			IF	(((bScrew1Found OR (bScrew1MinFound AND lrPackageThreadTimes = 1)) AND mcScrewer1Stop.Done) OR NOT bRun1 OR mcScrewer1MoveRelative.Done) AND
				(((bScrew2Found OR (bScrew2MinFound AND lrPackageThreadTimes = 1)) AND mcScrewer2Stop.Done) OR NOT bRun2 OR mcScrewer2MoveRelative.Done)
			THEN
				 mcScrewer1MoveRelative.Execute 	:=	FALSE;
				 mcScrewer1Stop.Execute				:=	FALSE;
				 mcScrewer2MoveRelative.Execute 	:=	FALSE;		
				 mcScrewer2Stop.Execute				:=	FALSE;	 
				 iFindingScrewCASE					:=	iFindingScrewCASE	+	10;	
			END_IF
			
		50: 
			IF tonFindingScrewDelay.Q THEN
 				iFindingScrewCASE					:=	iFindingScrewCASE	+	10;						
			END_IF

		60:
			lrStartPosition1						:=	Screwing1AxisRef.NcToPlc.ActPos;
			lrStartPosition2						:=	Screwing2AxisRef.NcToPlc.ActPos;
			iFindingScrewCASE 						:=	0;
			eRunningState							:=	E_GripperScrewer.eScrewing;
			IF bOptionFindScrewInPushingPosition THEN // Opcja - szukanie gwintu w pozycji docisku
				// Przejście do pozycji zakręcania, dlatego że był w pozycji docisku
				eRunningState							:=	E_GripperScrewer.eToScrewingPosition;
			END_IF
		END_CASE
END_IF
END_ACTION

ACTION Running6ScrewingMomentaryMode:
				(********** TRYB MOMENTOWY **********)
					CASE iScrewingCase OF 	
					0:
						(* Wersja 2 - gearowanie Multi Master***************************************************************) 
						IF iTool <> 2 THEN
							bGripper1Actuator						:=	bRun1; // Ponowne załączanie chwytaków, dlatego
							bGripper2Actuator						:=	bRun2; // że jest możliwa duża ilość opcji
						ELSE
							bGripper1Actuator						:=	FALSE; // Ponowne załączanie chwytaków, dlatego
							bGripper2Actuator						:=	FALSE;
						END_IF
						mcHeightGearInMultiMaster.Enable			:=	TRUE;				
						(* Start zakręcania *)
						IF	mcHeightGearInMultiMaster.InGear AND 
							(tonGripper1Delay.Q OR sTool = 'ksztaltowa/do kulek' OR NOT bRun1) AND (tonGripper2Delay.Q OR sTool = 'ksztaltowa/do kulek'  OR NOT bRun2) // ton'y powinny być już wczesniej załączone jeżeli były chwytaki	
						THEN

							mcScrewer1TorqueControl.Execute					:=	bRun1;
							mcScrewer1TorqueControl.Torque					:=	5000;//(INT_TO_UINT(iScrewer1SetTorque+3)*10)+iScrewer1AddTorque;	
							mcScrewer1TorqueControl.TorqueRamp				:=	4000;
							mcScrewer1TorqueControl.VelocityLimitHigh		:=	10;							
							mcScrewer1TorqueControl.VelocityLimitLow		:=	-5000;//(lrScrewerSpeed);
												
							mcScrewer2TorqueControl.Execute					:=	bRun2;
							mcScrewer2TorqueControl.Torque					:=	5000;//(INT_TO_UINT(iScrewer2SetTorque+3)*10)+iScrewer2AddTorque;	
							mcScrewer2TorqueControl.TorqueRamp				:=	4000;
							mcScrewer2TorqueControl.VelocityLimitHigh		:=	10;							
							mcScrewer2TorqueControl.VelocityLimitLow		:=	-5000;//(lrScrewerSpeed);
	
							iScrewingCase									:=	iScrewingCase + 10;			
						END_IF
						
					10:	
					
						IF ABS(ABS(lrStartPosition1)-ABS(Screwing1AxisRef.NcToPlc.ActPos))>(lrPackageTurnoversToFullScrewed*360.0/7)  THEN 
							mcScrewer1TorqueControl.Torque					:=	-9;		
							mcScrewer1TorqueControl.TorqueRamp				:=	1500;					
							mcScrewer1TorqueControl.VelocityLimitLow		:=	-4000;
						END_IF	
							
						IF ABS(ABS(lrStartPosition2)-ABS(Screwing2AxisRef.NcToPlc.ActPos))>(lrPackageTurnoversToFullScrewed*360.0/7)  THEN 
							mcScrewer2TorqueControl.Torque					:=	-9;		
							mcScrewer2TorqueControl.TorqueRamp				:=	1500;					
							mcScrewer2TorqueControl.VelocityLimitLow		:=	-4000;
						END_IF	
						
						IF ABS(ABS(lrStartPosition1)-ABS(Screwing1AxisRef.NcToPlc.ActPos))>(lrPackageTurnoversToFullScrewed*360.0/6)  THEN 
							mcScrewer1TorqueControl.Torque					:=	(INT_TO_UINT(iScrewer1SetTorque)+iScrewer1AddTorque);		
							mcScrewer1TorqueControl.TorqueRamp				:=	4000;					
							mcScrewer1TorqueControl.VelocityLimitLow		:=	-(lrScrewerSpeed);
						END_IF	
							
						IF ABS(ABS(lrStartPosition2)-ABS(Screwing2AxisRef.NcToPlc.ActPos))>(lrPackageTurnoversToFullScrewed*360.0/6)  THEN 
							mcScrewer2TorqueControl.Torque					:=	(INT_TO_UINT(iScrewer2SetTorque)+iScrewer2AddTorque);		
							mcScrewer2TorqueControl.TorqueRamp				:=	4000;					
							mcScrewer2TorqueControl.VelocityLimitLow		:=	-(lrScrewerSpeed);
						END_IF						
						(*IF tonMomentaryScrewing1Timer.Q OR bWarning1 THEN
							mcScrewer1Stop.Execute				:=	TRUE;
							bGripper1Actuator					:=	FALSE;
							mcScrewer1TorqueControl.Execute		:=	FALSE;
							uiScrewing1TorqueControl			:=	0;
							bScrewed1							:=	TRUE;	
						END_IF
						IF tonMomentaryScrewing2Timer.Q OR bWarning2 THEN
							mcScrewer2Stop.Execute				:=	TRUE;
							bGripper2Actuator					:=	FALSE;
							mcScrewer2TorqueControl.Execute		:=	FALSE;
							uiScrewing2TorqueControl			:=	0;
							bScrewed2							:=	TRUE;		
						END_IF*)
								
						IF tonMomentaryScrewing1Timer.Q OR bWarning1 THEN
							bGripper1Actuator					:=	FALSE;
							bScrewed1							:=	TRUE;	
						END_IF
						IF tonMomentaryScrewing2Timer.Q OR bWarning2 THEN
							bGripper2Actuator					:=	FALSE;
							bScrewed2							:=	TRUE;		
						END_IF
				
						IF tonTightScrewing1TimerAndOpenedGripper.Q OR bWarning1 THEN
							mcScrewer1Stop.Execute				:=	TRUE;
							mcScrewer1TorqueControl.Execute		:=	FALSE;
						END_IF
						IF tonTightScrewing2TimerAndOpenedGripper.Q OR bWarning2 THEN
							mcScrewer2Stop.Execute				:=	TRUE;
							mcScrewer2TorqueControl.Execute		:=	FALSE;
						END_IF											
				
						// Warunki zakręcenia zaleznie od uruchomionej zakręcarki
//						IF (bScrewed1 OR NOT bRun1) AND (bScrewed2 OR NOT bRun2) AND
//							(mcScrewer1Stop.Done OR NOT mcScrewer1Stop.Execute) AND 
//							(mcScrewer2Stop.Done OR NOT mcScrewer2Stop.Execute) THEN
						IF (tonTightScrewing1TimerAndOpenedGripper.Q OR NOT bRun1) AND (tonTightScrewing2TimerAndOpenedGripper.Q OR NOT bRun2) AND
							(mcScrewer1Stop.Done OR NOT mcScrewer1Stop.Execute) AND 
							(mcScrewer2Stop.Done OR NOT mcScrewer2Stop.Execute) THEN
								mcScrewer1Stop.Execute			:= FALSE;
								mcScrewer2Stop.Execute			:= FALSE;
								iScrewingCase					:= iScrewingCase + 10;		
						END_IF
					20:
						(* Rozgearowanie osi *)
						mcHeightGearOut.Execute				:=	TRUE;
						mcHeightGearInMultiMaster.Enable	:=	FALSE;
	
						IF  mcHeightGearOut.Done THEN
							mcHeightGearOut.Execute					:= FALSE;
							eRunningState							:= E_GripperScrewer.eHolding;	
							iScrewingCase							:= 0;	
						END_IF			
					END_CASE
END_ACTION

ACTION Running6ScrewingPositionTorqueMode:
				(********* TRYB POZYCYJNY  *********)
				
				lrPackageThreadPitch;	
				(*Wymuszanie zwiększonego momentu przez 1/4 całego zakręcania*)
				IF ABS(ABS(lrStartPosition1)-ABS(Screwing1AxisRef.NcToPlc.ActPos))>(lrPackageTurnoversToFullScrewed*360.0/7)  THEN 
							uiScrewing1TorqueControl			:=	(INT_TO_UINT(iScrewer1SetTorque+3)*10)+(iScrewer1AddTorque*10);	
				ELSE		uiScrewing1TorqueControl			:=	6000;
				END_IF
				//uiScrewing1TorqueControl			:=	(INT_TO_UINT(iScrewerSetTorque+3)*10)+iScrewer1AddTorque;	
				(*Wymuszanie zwiększonego momentu przez 1/4 całego zakręcania*)
				IF ABS(ABS(lrStartPosition2)-ABS(Screwing2AxisRef.NcToPlc.ActPos))>(lrPackageTurnoversToFullScrewed*360.0/7)  THEN 
							uiScrewing2TorqueControl			:=	(INT_TO_UINT(iScrewer2SetTorque+3)*10)+(iScrewer2AddTorque*10);		
				ELSE		uiScrewing2TorqueControl			:=	6000;
				END_IF	

					CASE iScrewingCase OF 	
					0:
						(* Wersja 2 - gearowanie Multi Master***************************************************************) 
						IF iTool <> 2 THEN
							bGripper1Actuator						:=	bRun1; // Ponowne załączanie chwytaków, dlatego
							bGripper2Actuator						:=	bRun2; // że jest możliwa duża ilość opcji
						ELSE
							bGripper1Actuator						:=	FALSE; // Ponowne załączanie chwytaków, dlatego
							bGripper2Actuator						:=	FALSE; // że jest możliwa duża ilość opcji
						END_IF
						mcHeightGearInMultiMaster.Enable			:=	TRUE;				
						(* Start zakręcania *)
						IF	mcHeightGearInMultiMaster.InGear AND 
							(tonGripper1Delay.Q OR sTool = 'ksztaltowa/do kulek' OR NOT bRun1) AND (tonGripper2Delay.Q OR sTool = 'ksztaltowa/do kulek' OR NOT bRun2) // ton'y powinny być już wczesniej załączone jeżeli były chwytaki	
						THEN

							CASE iScrewing2Case OF 	
								
							0:
							
								mcScrewer1MoveVelocity2.Velocity		:=	5000;
								mcScrewer1MoveVelocity2.Execute		:=	bRun1;
								mcScrewer1MoveVelocity2.Direction	:=	MC_Positive_Direction;
																				
								mcScrewer2MoveVelocity2.Velocity		:=	5000;
								mcScrewer2MoveVelocity2.Execute		:=	bRun2;
								mcScrewer2MoveVelocity2.Direction	:=	MC_Positive_Direction;	
	
								iScrewing2Case						:=	iScrewing2Case + 10;										
							
							10:
								mcScrewer1MoveVelocity2.Execute		:=	FALSE;
								mcScrewer2MoveVelocity2.Execute		:=	FALSE;
							
								iScrewing2Case						:=	iScrewing2Case + 10;
	
							20:
							
								mcScrewer1MoveVelocity.Velocity		:=	lrScrewerSpeed;		
								mcScrewer1MoveVelocity.Direction	:=	MC_Positive_Direction;	
								IF ABS(ABS(lrStartPosition1)-ABS(Screwing1AxisRef.NcToPlc.ActPos))>(lrPackageTurnoversToFullScrewed*360.0/7)  THEN 									
									mcScrewer1MoveVelocity.Execute		:=	bRun1;									
								END_IF
								mcScrewer2MoveVelocity.Velocity		:=	lrScrewerSpeed;	
								mcScrewer1MoveVelocity.Direction		:=	MC_Positive_Direction;	
								IF ABS(ABS(lrStartPosition2)-ABS(Screwing2AxisRef.NcToPlc.ActPos))>(lrPackageTurnoversToFullScrewed*360.0/7)  THEN 
	
									mcScrewer2MoveVelocity.Execute		:=	bRun2;
								END_IF			

								IF (mcScrewer1MoveVelocity.Execute OR NOT bRun1) AND (mcScrewer2MoveVelocity.Execute OR NOT bRun2) THEN
									iScrewing2Case					:= 0	;
									iScrewingCase					:= iScrewingCase + 10;		
								END_IF
								
							END_CASE
							
						END_IF
						
					10:	
					
						(*Zmniejszanie prędkości jeżeli jest już przytrzymanie*)
						IF tonTightScrewing1Timer.ET > T#0S AND Screwing1AxisRef.NcToPlc.ActVelo < 10 THEN
							//mcScrewer1MoveVelocity.Execute		:= FALSE;
							//mcScrewer1MoveVelocity2.Execute		:= FALSE;
							
							//mcScrewer1MoveVelocity3.Velocity	:=	10;
							//mcScrewer1MoveVelocity3.Execute		:=	bRun1;
							//mcScrewer1MoveVelocity3.Direction	:=	MC_Positive_Direction;		

							rScrewing1ProportionalGain	:= 0;
							//rScrewing2ProportionalGain	:= 0;												
						END_IF
						
						IF tonTightScrewing2Timer.ET > T#0S AND Screwing2AxisRef.NcToPlc.ActVelo < 10 THEN
							//mcScrewer2MoveVelocity.Execute		:= FALSE;
							//mcScrewer2MoveVelocity2.Execute		:= FALSE;
							
							//mcScrewer2MoveVelocity3.Velocity	:=	10;
							//mcScrewer2MoveVelocity3.Execute		:=	bRun1;
							//mcScrewer2MoveVelocity3.Direction	:=	MC_Positive_Direction;		

							//rScrewing1ProportionalGain	:= 0;
							rScrewing2ProportionalGain	:= 0;												
						END_IF					
					
						(* Sprawdzanie czy osiągnięto moment lub zbyt długie zakracanie*)				
						IF tonTightScrewing1Timer.Q OR bWarning1 THEN
							bGripper1Actuator					:=	FALSE;
							bScrewed1							:=	TRUE;	
						END_IF
						IF tonTightScrewing2Timer.Q OR bWarning2 THEN
							bGripper2Actuator					:=	FALSE;
							bScrewed2							:=	TRUE;		
						END_IF
	
						IF tonTightScrewing1TimerAndOpenedGripper.Q THEN
							mcScrewer1Stop.Execute				:=	TRUE;
							mcScrewer1MoveVelocity.Execute		:=	FALSE;
							mcScrewer1MoveVelocity2.Execute		:=	FALSE;
							mcScrewer1MoveVelocity3.Execute		:=	FALSE;							
							uiScrewing1TorqueControl			:=	0;
						END_IF
						IF tonTightScrewing2TimerAndOpenedGripper.Q THEN
							mcScrewer2Stop.Execute				:=	TRUE;
							mcScrewer2MoveVelocity.Execute		:=	FALSE;
							mcScrewer2MoveVelocity2.Execute		:=	FALSE;	
							mcScrewer2MoveVelocity3.Execute		:=	FALSE;							
							uiScrewing2TorqueControl			:=	0;
						END_IF
					
						// Warunki zakręcenia zaleznie od uruchomionej zakręcarki
						IF (tonTightScrewing1TimerAndOpenedGripper.Q OR NOT bRun1) AND (tonTightScrewing2TimerAndOpenedGripper.Q OR NOT bRun2) AND
							(mcScrewer1Stop.Done OR NOT mcScrewer1Stop.Execute) AND 
							(mcScrewer2Stop.Done OR NOT mcScrewer2Stop.Execute) THEN
								mcScrewer1Stop.Execute			:= FALSE;
								mcScrewer2Stop.Execute			:= FALSE;
								iScrewingCase					:= iScrewingCase + 10;		
						END_IF
						
					20:
						(* Rozgearowanie osi *)
						mcHeightGearOut.Execute				:=	TRUE;
						mcHeightGearInMultiMaster.Enable	:=	FALSE;
	
						IF  mcHeightGearOut.Done THEN
							mcHeightGearOut.Execute					:= FALSE;
							eRunningState							:= E_GripperScrewer.eHolding;	
							iScrewingCase							:= 0;	
						END_IF			
					END_CASE
END_ACTION

ACTION Screwer1ControlBlocks:
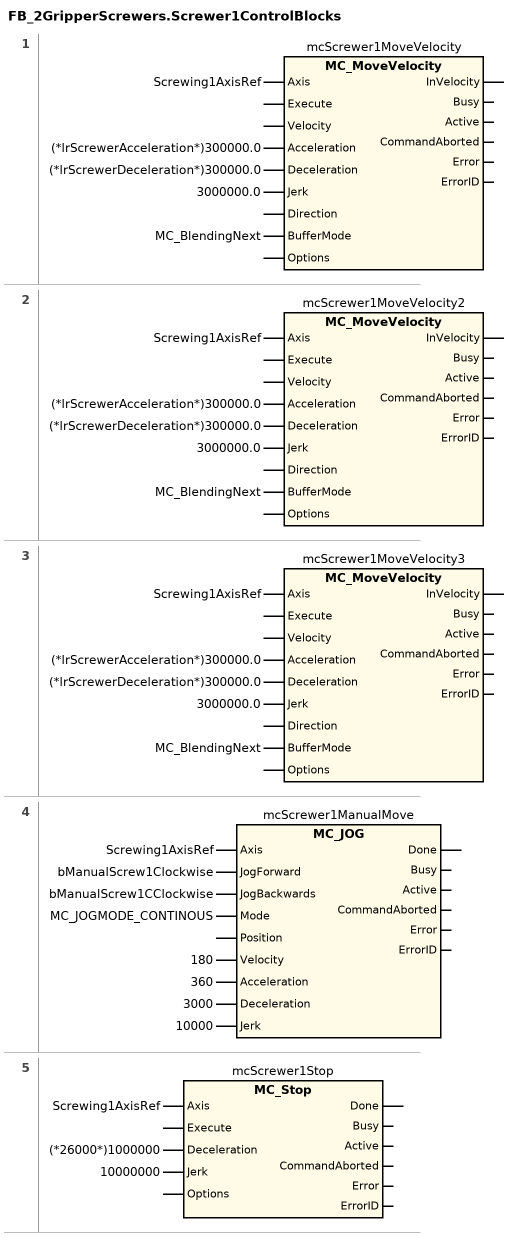
// NETWORK 1
mcScrewer1MoveVelocity(
    Axis := Screwing1AxisRef,
    Acceleration := (*lrScrewerAcceleration*)300000.0,
    Deceleration := (*lrScrewerDeceleration*)300000.0,
    Jerk := 3000000.0,
    BufferMode := MC_BlendingNext); // MC_MoveVelocity

// NETWORK 2
mcScrewer1MoveVelocity2(
    Axis := Screwing1AxisRef,
    Acceleration := (*lrScrewerAcceleration*)300000.0,
    Deceleration := (*lrScrewerDeceleration*)300000.0,
    Jerk := 3000000.0,
    BufferMode := MC_BlendingNext); // MC_MoveVelocity

// NETWORK 3
mcScrewer1MoveVelocity3(
    Axis := Screwing1AxisRef,
    Acceleration := (*lrScrewerAcceleration*)300000.0,
    Deceleration := (*lrScrewerDeceleration*)300000.0,
    Jerk := 3000000.0,
    BufferMode := MC_BlendingNext); // MC_MoveVelocity

// NETWORK 4
mcScrewer1ManualMove(
    Axis := Screwing1AxisRef,
    JogForward := bManualScrew1Clockwise,
    JogBackwards := bManualScrew1CClockwise,
    Mode := MC_JOGMODE_CONTINOUS,
    Velocity := 180,
    Acceleration := 360,
    Deceleration := 3000,
    Jerk := 10000); // MC_JOG

// NETWORK 5
mcScrewer1Stop(Axis := Screwing1AxisRef, Deceleration := (*26000*)1000000, Jerk := 10000000); // MC_Stop

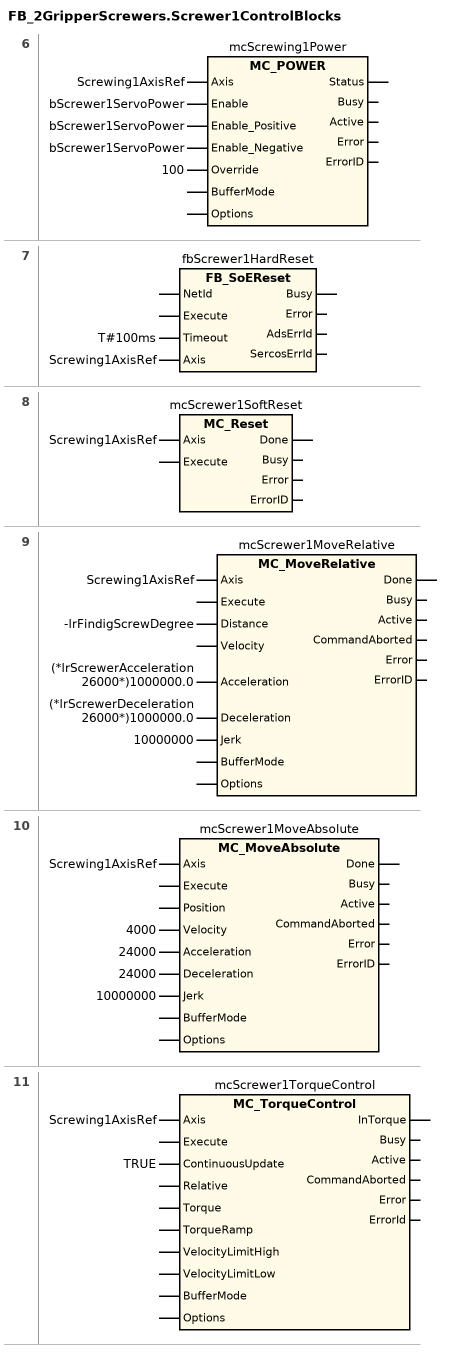
// NETWORK 6
mcScrewing1Power(
    Axis := Screwing1AxisRef,
    Enable := bScrewer1ServoPower,
    Enable_Positive := bScrewer1ServoPower,
    Enable_Negative := bScrewer1ServoPower,
    Override := 100); // MC_POWER

// NETWORK 7
fbScrewer1HardReset(Timeout := T#100ms, Axis := Screwing1AxisRef); // FB_SoEReset

// NETWORK 8
mcScrewer1SoftReset(Axis := Screwing1AxisRef); // MC_Reset

// NETWORK 9
mcScrewer1MoveRelative(
    Axis := Screwing1AxisRef,
    Distance := -lrFindigScrewDegree,
    Acceleration := (*lrScrewerAcceleration 26000*)1000000.0,
    Deceleration := (*lrScrewerDeceleration 26000*)1000000.0,
    Jerk := 10000000); // MC_MoveRelative

// NETWORK 10
mcScrewer1MoveAbsolute(
    Axis := Screwing1AxisRef,
    Velocity := 4000,
    Acceleration := 24000,
    Deceleration := 24000,
    Jerk := 10000000); // MC_MoveAbsolute

// NETWORK 11
mcScrewer1TorqueControl(Axis := Screwing1AxisRef, ContinuousUpdate := TRUE); // MC_TorqueControl

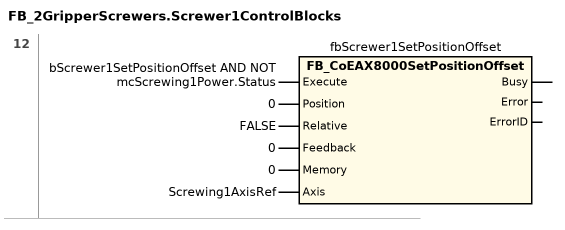
// NETWORK 12
fbScrewer1SetPositionOffset(
    Execute := bScrewer1SetPositionOffset AND NOT mcScrewing1Power.Status,
    Position := 0,
    Relative := FALSE,
    Feedback := 0,
    Memory := 0,
    Axis := Screwing1AxisRef); // FB_CoEAX8000SetPositionOffset
END_ACTION

ACTION Screwer2ControlBlocks:
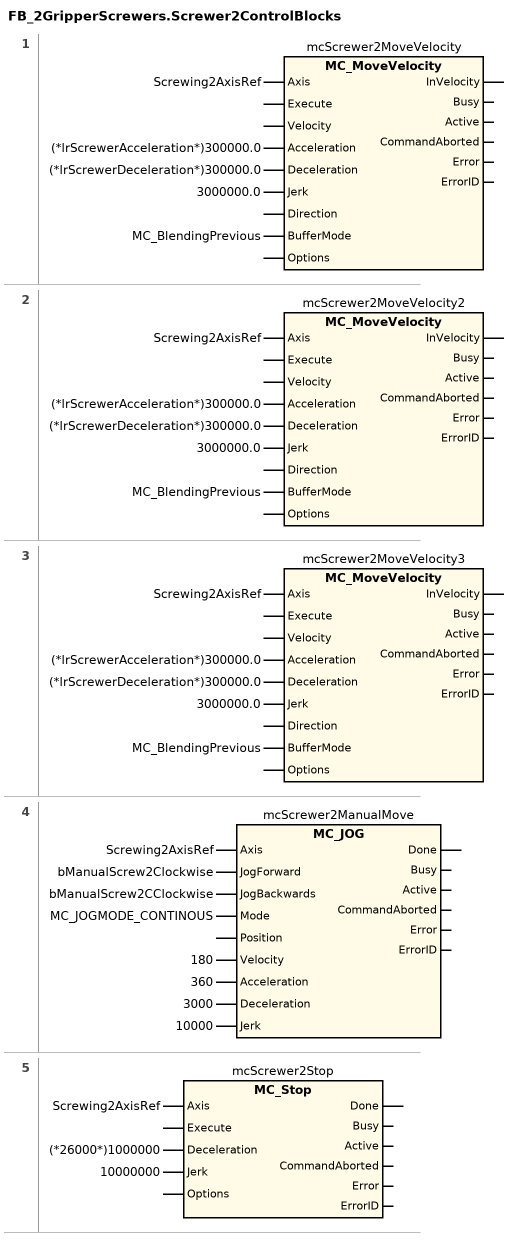
// NETWORK 1
mcScrewer2MoveVelocity(
    Axis := Screwing2AxisRef,
    Acceleration := (*lrScrewerAcceleration*)300000.0,
    Deceleration := (*lrScrewerDeceleration*)300000.0,
    Jerk := 3000000.0,
    BufferMode := MC_BlendingPrevious); // MC_MoveVelocity

// NETWORK 2
mcScrewer2MoveVelocity2(
    Axis := Screwing2AxisRef,
    Acceleration := (*lrScrewerAcceleration*)300000.0,
    Deceleration := (*lrScrewerDeceleration*)300000.0,
    Jerk := 3000000.0,
    BufferMode := MC_BlendingPrevious); // MC_MoveVelocity

// NETWORK 3
mcScrewer2MoveVelocity3(
    Axis := Screwing2AxisRef,
    Acceleration := (*lrScrewerAcceleration*)300000.0,
    Deceleration := (*lrScrewerDeceleration*)300000.0,
    Jerk := 3000000.0,
    BufferMode := MC_BlendingPrevious); // MC_MoveVelocity

// NETWORK 4
mcScrewer2ManualMove(
    Axis := Screwing2AxisRef,
    JogForward := bManualScrew2Clockwise,
    JogBackwards := bManualScrew2CClockwise,
    Mode := MC_JOGMODE_CONTINOUS,
    Velocity := 180,
    Acceleration := 360,
    Deceleration := 3000,
    Jerk := 10000); // MC_JOG

// NETWORK 5
mcScrewer2Stop(Axis := Screwing2AxisRef, Deceleration := (*26000*)1000000, Jerk := 10000000); // MC_Stop

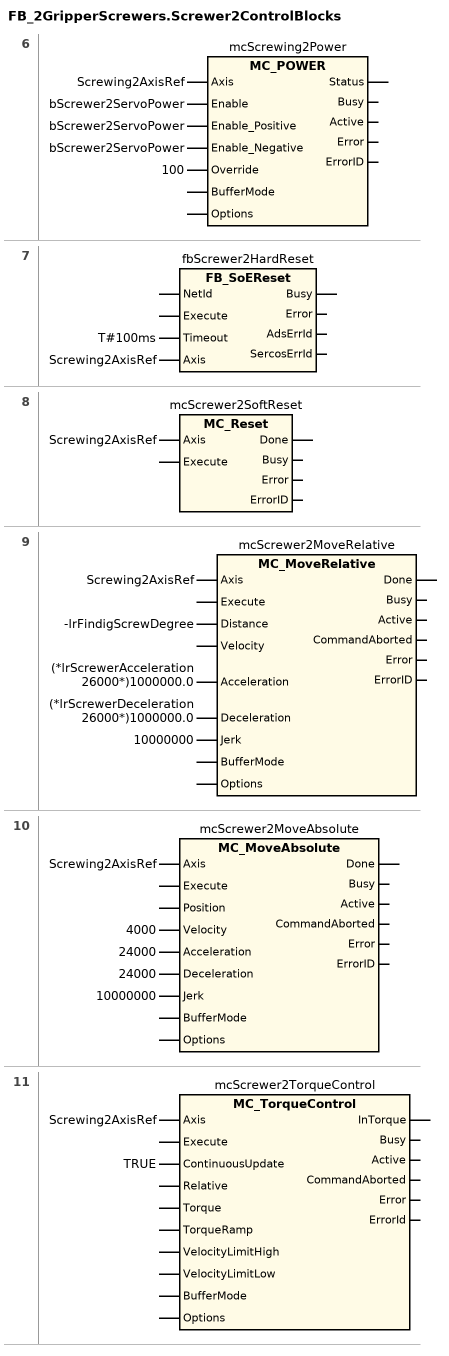
// NETWORK 6
mcScrewing2Power(
    Axis := Screwing2AxisRef,
    Enable := bScrewer2ServoPower,
    Enable_Positive := bScrewer2ServoPower,
    Enable_Negative := bScrewer2ServoPower,
    Override := 100); // MC_POWER

// NETWORK 7
fbScrewer2HardReset(Timeout := T#100ms, Axis := Screwing2AxisRef); // FB_SoEReset

// NETWORK 8
mcScrewer2SoftReset(Axis := Screwing2AxisRef); // MC_Reset

// NETWORK 9
mcScrewer2MoveRelative(
    Axis := Screwing2AxisRef,
    Distance := -lrFindigScrewDegree,
    Acceleration := (*lrScrewerAcceleration 26000*)1000000.0,
    Deceleration := (*lrScrewerDeceleration 26000*)1000000.0,
    Jerk := 10000000); // MC_MoveRelative

// NETWORK 10
mcScrewer2MoveAbsolute(
    Axis := Screwing2AxisRef,
    Velocity := 4000,
    Acceleration := 24000,
    Deceleration := 24000,
    Jerk := 10000000); // MC_MoveAbsolute

// NETWORK 11
mcScrewer2TorqueControl(Axis := Screwing2AxisRef, ContinuousUpdate := TRUE); // MC_TorqueControl

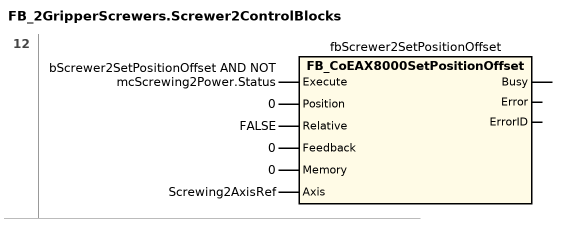
// NETWORK 12
fbScrewer2SetPositionOffset(
    Execute := bScrewer2SetPositionOffset AND NOT mcScrewing2Power.Status,
    Position := 0,
    Relative := FALSE,
    Feedback := 0,
    Memory := 0,
    Axis := Screwing2AxisRef); // FB_CoEAX8000SetPositionOffset
END_ACTION

ACTION Simulation:
(* Przyśpieszanie bloku gdy jest włączona symulacja*)

//tonSimulationScrewing1			(IN:=eRunningState=E_GripperScrewer.eScrewing 	AND bRun1 AND NOT bScrewed1 AND bSimulation,	PT:=T#0MS);
//tonSimulationScrewing2			(IN:=eRunningState=E_GripperScrewer.eScrewing 	AND bRun1 AND NOT bScrewed2 AND bSimulation,	PT:=T#0MS);

IF bSimulation THEN 			// Włączona symulacja
	tTooLongScrewing1 := T#250MS;
	tTooLongScrewing2 := T#250MS;	
ELSE							// Normalna praca
	tTooLongScrewing1 := T#3S; 	//Zmienić na 2
	tTooLongScrewing2 := T#3S;	//Zmienić na 2
END_IF
END_ACTION

ACTION Statistics:

IF LREAL_TO_INT(lrHeightEndScrewingPosition)<> LREAL_TO_INT(lrHeightReadyPosition) THEN
	rtrigCycleTimerRead(CLK:=LREAL_TO_INT(lrHeightActualPosition) = LREAL_TO_INT(lrHeightReadyPosition));
	IF rtrigCycleTimerRead.Q THEN
			tCycleTime:=tonCycleTimer.ET;
	END_IF
	tonCycleTimer(IN:=LREAL_TO_INT(lrHeightActualPosition) <> LREAL_TO_INT(lrHeightReadyPosition),PT:=T#1D);	
ELSE
	rtrigCycleTimerRead(CLK:=(eRunningState=E_GripperScrewer.eDone) OR (eRunningState=E_GripperScrewer.eNotDone));
	IF rtrigCycleTimerRead.Q THEN
		tCycleTime:=tonCycleTimer.ET;
	END_IF
	tonCycleTimer(IN:=eRunningState>E_GripperScrewer.eReady,PT:=T#1D);
END_IF
END_ACTION

ACTION Tools:
(*Narzędzia*)
AsToolDescription[0] := 'Głowica dwuszczękowa';
AsToolDescription[1] := 'Głowica trójszczękowa'; 
AsToolDescription[2] := 'Głowica kształtowa/do kulek';
AsToolDescription[3] := 'Głowica wbijająca'; 
AsToolDescription[4] := 'Głowica zasysająca';


(*Głowica wbijająca*)
IF iTool = 3 THEN
	bOptionCapPushingWithoutScrewing := TRUE;
ELSE
	bOptionCapPushingWithoutScrewing := FALSE;
END_IF

(*Przepisanie wybranego narzędzia do zmiennej typu string*)
(*!!!!! NIE ZMIENIAĆ OPISÓW, POWIĄZANE W PROGRAMIE !!!!!!*)
(* Wysokość narzędzia od pkt. bazowania

		Glowica dwuszczekowa
           |	|
		   |	|
	|------|    |-----|
	|	 _______	  |
	|	|		  |   |
   ||	||		  |   |
   ||	||		  |	  |
   |---- |		  -----	<-pkt. bazowania 	<-|
   |	 |	                                  |
   |	 ---|	  							iToolHeight (mm)
   |druk	|                                 |
   ---------|	  							<-|

*)


IF iTool = 0 THEN sTool := 'dwuszczekowa';			iToolHeight	:=	23;		END_IF 
IF iTool = 1 THEN sTool := 'trojszczekowa';			iToolHeight	:=	-5;	END_IF 
IF iTool = 2 THEN sTool := 'ksztaltowa/do kulek';	iToolHeight	:=	-5;		END_IF 
IF iTool = 3 THEN sTool := 'wbijajaca';				iToolHeight	:=	23;		END_IF 
IF iTool = 4 THEN sTool := 'zasysajaca';			iToolHeight	:=	-4;		END_IF
END_ACTION

ACTION TorqueControl:

(*Konfiguracja MC_TorqueControl*)
//T_TorqueControlOptions;
mcScrewer1TorqueControl.Options.EnableManualTorqueStartValue := TRUE;
mcScrewer1TorqueControl.Options.ManualTorqueStartValue       := Screwing1AxisRef.NcToPlc.ActTorque;

mcScrewer2TorqueControl.Options.EnableManualTorqueStartValue := TRUE;
mcScrewer2TorqueControl.Options.ManualTorqueStartValue       :=  Screwing2AxisRef.NcToPlc.ActTorque;
END_ACTION

ACTION Warnings:
//Resetowanie warningów przy nastepnym cyklu

IF rtRun1.Q  OR rtRun2.Q THEN
	
	bWarning1			:=	FALSE;
	bWarning1A			:=	FALSE;
	bWarning1B			:=	FALSE;
	bWarning1C			:=	FALSE;
	bWarning1D			:=	FALSE;
	bWarning1E			:=	FALSE;	
	bWarning2			:=	FALSE;
	bWarning2A			:=	FALSE;
	bWarning2B			:=	FALSE;
	bWarning2C			:=	FALSE;
	bWarning2D			:=	FALSE;
	bWarning2E			:=	FALSE;
END_IF
END_ACTION

END_FUNCTION_BLOCK

// ---- POUs/FB/POUsAxisOnline/AX8000/FB_McAxisOnlineAX8000.TcPOU
//==================================================================================================
//							Beckhoff Automation Poland
//									7.12.2018
//	Wszystkomajacy blok funkcyjny do sterowania osia, 
//	wymagane biblioteki: Tc2_EtherCAT, Tc2_MC2_Drive, Tc2_MC2
//  v1.5	|| TC v 3.1.4022.27		|| - dodane opisy bledow w formie zmiennych typu string
// 	v1.4 	|| TC v 3.1.4022.20	 	|| - ACT_MotorMonitoring - only for real axis
// 	v1.3 	|| TC v 3.1.4022.16	 	|| - spojne z AX5000
// 	v1.2 	|| TC v 3.1.4022.16	 	|| - Added ACT_SetPositionIO, migration part of logic from ACT_SetPosition to ACT_SetPositionIO
// 	v1.1 	|| TC v 3.1.4022.16	 	|| - ACT_MotorMonitoring - is executing always, ACT_Initialization - optimalization
// 	v1.0 	|| TC v 3.1.4022.16	 	|| - first edition
//==================================================================================================
{attribute 'reflection'}
FUNCTION_BLOCK FB_McAxisOnlineAX8000
VAR_IN_OUT
	stMcAxisOnline						: ST_McAxisOnline;
	Axis								: AXIS_REF;
END_VAR
VAR
	mcPower								: MC_Power;
	mcStop								: MC_Stop;
	mcHalt								: MC_Halt;
	mcStopSS1							: MC_Stop;
	mcStopSS2							: MC_Stop;
	mcReset								: MC_Reset;
	mcHome								: MC_Home;
	mcSetPosition						: MC_SetPosition;
	fbSetPositionOffset					: FB_CoEAX8000SetPositionOffset;
	mcJog								: MC_Jog;

	mcMoveAbsolute						: MC_MoveAbsolute;
	mcMoveRelative						: MC_MoveRelative;
	mcMoveVelocity						: MC_MoveVelocity;
	mcMoveModulo						: MC_MoveModulo;
	mcMoveAbsolute2						: MC_MoveAbsolute;
	mcMoveRelative2						: MC_MoveRelative;
	mcMoveVelocity2						: MC_MoveVelocity;
	mcMoveModulo2						: MC_MoveModulo;

	fbMotorMonitoring					: FB_MotorMonitoringAX8000;
	fbHoldingBrakeCtrl					: FB_HoldingBrakeCtrlAX8000;
	fbNcLimitSwitch						: FB_NcSWLimitSwitchCtrl;
	tonGetDriveDiag						: TON;
	fbReadChannelErrorCode				: FB_ReadChannelErrorCodeAX8000;
	
	mcReadDriveAddress					: MC_ReadDriveAddress;
	mcReadParameterSet					: MC_ReadParameterSet;
	fbGetDriveRef						: FB_GetDriveRef;

	// Internal
	bInitialized						: BOOL;
	bCommError							: BOOL;
	bReadParameterError					: BOOL;
	bInitError							: BOOL;
	bDriveError							: BOOL;
	bFBError							: BOOL;
	
// Initialization
	iInitStep							: INT;
	bInitializationError				: BOOL;
	wInitializationErrorCounter			: WORD;
	bDriveAddressReady					: BOOL;
	bDriveRefReady						: BOOL;
	bReadParameterSetReady				: BOOL;
	tonDelay							: TON;
// Re init
	udiOnlineChangeCntOld				: UDINT;
	bOnlineChangeDetected				: BOOL;
	bReInit								: BOOL;
	bReInitialized						: BOOL;
	bReInitializationError				: BOOL;
	{attribute 'instance-path'}
	{attribute 'noinit'}
	sInstancePath						: STRING;
END_VAR

// Device dependent initialization 
ACT_Initialization();
// Device independent commands, mostly NC 
ACT_States();
ACT_SWLimitSwitch();
ACT_Stop();
ACT_Power();
ACT_Homing();
ACT_Jog();
ACT_Move();
ACT_Reset();
ACT_SetPosition();
// Device dependent commands
// Motor monitoring possible only with real axis
IF NOT Axis.Status.OpMode.SimulationAxis THEN
	ACT_MotorMonitoring();
END_IF
// Device dependent commands, possible only on real axis after complete initialization
IF bInitialized AND NOT Axis.Status.OpMode.SimulationAxis THEN
	ACT_SetPositionIO();
	ACT_DriveDiag();
	ACT_HoldingBrakeCtrl();
END_IF

// Device independent error collection
ACT_ErrorCollection();

ACTION ACT_DriveDiag:
// Auto update when drive error
tonGetDriveDiag(IN:= stMcAxisOnline.stError.bDriveError AND NOT tonGetDriveDiag.Q, PT:= T#5S, Q=> , ET=> );

fbReadChannelErrorCode(	bExecute				:= stMcAxisOnline.stChannelErrorCode.bExecute OR tonGetDriveDiag.Q,
						stDriveRef				:= stMcAxisOnline.stDriveRef,
						bBusy					=> stMcAxisOnline.stChannelErrorCode.bBusy,
						bError					=> stMcAxisOnline.stChannelErrorCode.bError,
						iAdsErrId				=> stMcAxisOnline.stChannelErrorCode.uiAdsErrId,
						iCANopenErrId			=> stMcAxisOnline.stChannelErrorCode.uiSecErrId,
						uiChannelErrorCode		=> stMcAxisOnline.stChannelErrorCode.uiChannelErrorCode,
						uiChannelErrorCodeHex	=> stMcAxisOnline.stChannelErrorCode.uiChannelErrorCodeHex);
END_ACTION

ACTION ACT_ErrorCollection:
// Error flags
stMcAxisOnline.stError.bDriveError					:= Axis.Status.DriveDeviceError;

stMcAxisOnline.stError.bNcError						:= Axis.Status.Error;

stMcAxisOnline.stError.bFBError						:= stMcAxisOnline.mcPower.bError OR stMcAxisOnline.mcReset.bError OR stMcAxisOnline.mcHome.bError OR stMcAxisOnline.mcJog.bError
													OR stMcAxisOnline.mcHalt.bError OR stMcAxisOnline.mcStop.bError OR stMcAxisOnline.mcSS1.bError OR stMcAxisOnline.mcSS2.bError
													OR stMcAxisOnline.mcMoveAbsolute.bError OR stMcAxisOnline.mcMoveRelative.bError OR stMcAxisOnline.mcMoveVelocity.bError OR stMcAxisOnline.mcMoveModulo.bError
													OR stMcAxisOnline.mcMoveAbsolute2.bError OR stMcAxisOnline.mcMoveRelative2.bError OR stMcAxisOnline.mcMoveVelocity2.bError OR stMcAxisOnline.mcMoveModulo2.bError
													OR stMcAxisOnline.stNcLimitSwitch.bError OR stMcAxisOnline.mcSetPosition.bError;
									
stMcAxisOnline.stError.bCommunicationError			:= stMcAxisOnline.stChannelErrorCode.bError OR stMcAxisOnline.stSetPositionOffset.bError OR stMcAxisOnline.stMotorMonitoring.bError OR stMcAxisOnline.stHoldingBrake.bError;

stMcAxisOnline.stError.bError						:= stMcAxisOnline.stError.bDriveError OR stMcAxisOnline.stError.bNcError OR stMcAxisOnline.stError.bFBError OR stMcAxisOnline.stError.bCommunicationError;
stMcAxisOnline.bError								:= stMcAxisOnline.stError.bError; // Forward one stage up

// Error codes
stMcAxisOnline.stError.uiDriveErrorID 				:= stMcAxisOnline.stChannelErrorCode.uiChannelErrorCode;
stMcAxisOnline.stError.uiDriveErrorIDHex 			:= stMcAxisOnline.stChannelErrorCode.uiChannelErrorCodeHex;

stMcAxisOnline.stError.udiNcErrorID 				:= Axis.Status.ErrorID;
stMcAxisOnline.stError.udiNcErrorIDHex 				:= Axis.Status.ErrorID;
	

stMcAxisOnline.stError.udiFBErrorID 				:= 	stMcAxisOnline.mcPower.udiErrorID + 
														stMcAxisOnline.mcReset.udiErrorID + 
														stMcAxisOnline.mcHome.udiErrorID + 
														stMcAxisOnline.mcJog.udiErrorID +
														stMcAxisOnline.mcHalt.udiErrorID + 
														stMcAxisOnline.mcStop.udiErrorID + 
														stMcAxisOnline.mcSS1.udiErrorID + 
														stMcAxisOnline.mcSS2.udiErrorID +
														stMcAxisOnline.mcMoveAbsolute.udiErrorID + 
														stMcAxisOnline.mcMoveRelative.udiErrorID + 
														stMcAxisOnline.mcMoveVelocity.udiErrorID + 
														stMcAxisOnline.mcMoveModulo.udiErrorID +
														stMcAxisOnline.mcMoveAbsolute2.udiErrorID + 
														stMcAxisOnline.mcMoveRelative2.udiErrorID + 
														stMcAxisOnline.mcMoveVelocity2.udiErrorID + 
														stMcAxisOnline.mcMoveModulo2.udiErrorID +
														stMcAxisOnline.stNcLimitSwitch.udiErrorID + 
														stMcAxisOnline.mcSetPosition.udiErrorID;

stMcAxisOnline.stError.udiFBErrorIDHex 				:= stMcAxisOnline.stError.udiFBErrorID;

stMcAxisOnline.stError.udiErrorID					:= stMcAxisOnline.stSetPositionOffset.udiErrorID;
stMcAxisOnline.stError.uiAdsErrorID					:= stMcAxisOnline.stChannelErrorCode.uiAdsErrId + stMcAxisOnline.stMotorMonitoring.uiAdsErrId + stMcAxisOnline.stHoldingBrake.uiAdsErrId;
stMcAxisOnline.stError.uiSecErrorID					:= stMcAxisOnline.stChannelErrorCode.uiSecErrId + stMcAxisOnline.stMotorMonitoring.uiSecErrId + stMcAxisOnline.stHoldingBrake.uiSecErrId;

stMcAxisOnline.stError.sNcError						:= F_AxErrMsg(stMcAxisOnline.stError.udiNcErrorID);
stMcAxisOnline.stError.sDriveError					:= F_AX8xErrMsg(stMcAxisOnline.stError.uiDriveErrorID);
END_ACTION

ACTION ACT_HoldingBrakeCtrl:
fbHoldingBrakeCtrl(	bForceLock			:= stMcAxisOnline.stHoldingBrake.bForceLock,
					bForceUnlock		:= stMcAxisOnline.stHoldingBrake.bForceUnlock,
					stDriveRef			:= stMcAxisOnline.stDriveRef,
					bBusy				=> stMcAxisOnline.stHoldingBrake.bBusy,
					bError				=> stMcAxisOnline.stHoldingBrake.bError,
					iAdsErrId			=> stMcAxisOnline.stHoldingBrake.uiAdsErrId,
					iCANopenErrId		=> stMcAxisOnline.stHoldingBrake.uiSecErrId);
END_ACTION

ACTION ACT_Homing:
mcHome(		Axis						:= Axis,
			Execute						:= stMcAxisOnline.mcHome.bExecute,
			Position					:= stMcAxisOnline.mcHome.lrPosition,
			HomingMode					:= stMcAxisOnline.mcHome.eHomingMode,
			BufferMode					:= stMcAxisOnline.mcHome.eBufferMode,
			Options						:= stMcAxisOnline.mcHome.stOptions,
			bCalibrationCam				:= stMcAxisOnline.mcHome.bCalibrationCam,
			Done						=> stMcAxisOnline.mcHome.bDone,
			Busy						=> stMcAxisOnline.mcHome.bBusy,
			Active						=> stMcAxisOnline.mcHome.bActive,
			CommandAborted				=> stMcAxisOnline.mcHome.bCommandAborted,
			Error						=> stMcAxisOnline.mcHome.bError,
			ErrorID						=> stMcAxisOnline.mcHome.udiErrorID);
END_ACTION

ACTION ACT_Initialization:
// bInitialized flag is set just once. 
// bReInitialized ise set each time we do online change or request reinit operation
// bDriveAddressReady, bReadParameterSetReady, bDriveRefReady - set just once after successed read

// Online change detection
bOnlineChangeDetected					:= udiOnlineChangeCntOld <> _AppInfo.OnlineChangeCnt;
udiOnlineChangeCntOld 					:= _AppInfo.OnlineChangeCnt;
// Reset init
IF bReInit OR bOnlineChangeDetected THEN
	iInitStep							:= 0;
END_IF

//Initialization process
CASE iInitStep OF
	0:	// Read Drive Address
		
		stMcAxisOnline.mcReadDriveAddress.bExecute	:=	 TRUE;
		iInitStep						:= iInitStep + 10;
		
	10: // Wait for data
	
		IF NOT stMcAxisOnline.mcReadDriveAddress.bBusy THEN
			stMcAxisOnline.mcReadDriveAddress.bExecute	:=	 FALSE;
			IF stMcAxisOnline.mcReadDriveAddress.bDone THEN
				iInitStep 				:= iInitStep + 10;
				bDriveAddressReady 		:= TRUE;
			ELSE
				iInitStep 				:= 1000;		// Error step
			END_IF
		END_IF
		
	20:	// Read Parameter Set
		
		stMcAxisOnline.mcReadParameterSet.bExecute		:=	 TRUE;
		iInitStep						:= iInitStep + 10;
		
	30: // Wait for data
	
		IF NOT stMcAxisOnline.mcReadParameterSet.bBusy THEN
			stMcAxisOnline.mcReadParameterSet.bExecute	:=	 FALSE;
			IF stMcAxisOnline.mcReadParameterSet.bDone THEN
				iInitStep 				:= iInitStep + 10;
				bReadParameterSetReady 	:= TRUE;
			ELSE
				iInitStep 				:= 1000;		// Error step
			END_IF
		END_IF	
	
	40:	// Get Drive Ref
		
		stMcAxisOnline.stGetDriveRef.bExecute		:=	 TRUE;
		iInitStep						:= iInitStep + 10;
		
	50: // Wait for data
	
		IF NOT stMcAxisOnline.stGetDriveRef.bBusy THEN
			stMcAxisOnline.stGetDriveRef.bExecute	:=	 FALSE;
			IF NOT stMcAxisOnline.stGetDriveRef.bError THEN
				iInitStep 				:= iInitStep + 10;
				bDriveRefReady 			:= TRUE;
			ELSE
				iInitStep 				:= 1000;		// Error step
			END_IF
		END_IF
	
	60: // Success - initialized flag, clear error
		bReInitialized					:= bInitialized;	// TRUE only when it's not first initialization e.g. online change
		bInitialized 					:= TRUE;
		bReInitializationError			:= FALSE;			// TRUE only when it's not first initialization e.g. online change
		bInitializationError			:= FALSE;
		iInitStep 						:= iInitStep + 10;
		
	70: // Idle
	
		;
		
	1000: // Error step
		wInitializationErrorCounter 	:= wInitializationErrorCounter + 1;
		IF wInitializationErrorCounter < 100 THEN
			iInitStep					:= iInitStep + 5;			// Go to delay
		ELSE
			bReInitializationError		:= bInitializationError;	// TRUE only when it's not first initialization e.g. online change
			bInitializationError		:= TRUE;
			bReInitialized				:= FALSE;
			iInitStep 					:= iInitStep + 10;
		END_IF

	1005: // Delay step
		tonDelay(IN:= TRUE, PT:= T#1S);
		IF tonDelay.Q THEN
			tonDelay(IN:= FALSE, PT:= T#1S);
			iInitStep					:= 0;
		END_IF
		
	1010: // Idle after error
		;
	
END_CASE

mcReadDriveAddress(	Axis				:= Axis,
					Execute				:= stMcAxisOnline.mcReadDriveAddress.bExecute,
					Done				=> stMcAxisOnline.mcReadDriveAddress.bDone,
					Busy				=> stMcAxisOnline.mcReadDriveAddress.bBusy,
					Error				=> stMcAxisOnline.mcReadDriveAddress.bError,
					ErrorID				=> stMcAxisOnline.mcReadDriveAddress.udiErrorID,
					DriveAddress		=> stMcAxisOnline.stDriveAddress);
				
mcReadParameterSet(	Parameter			:= stMcAxisOnline.stAxisParameter,
					Axis				:= Axis,
					Execute				:= stMcAxisOnline.mcReadParameterSet.bExecute,
					Done				=> stMcAxisOnline.mcReadParameterSet.bDone,
					Busy				=> stMcAxisOnline.mcReadParameterSet.bBusy,
					Error				=> stMcAxisOnline.mcReadParameterSet.bError,
					ErrorID				=> stMcAxisOnline.mcReadParameterSet.udiErrorID);
					
fbGetDriveRef(		bExecute			:= stMcAxisOnline.stGetDriveRef.bExecute,
					bBusy				=> stMcAxisOnline.stGetDriveRef.bBusy,
					bError				=> stMcAxisOnline.stGetDriveRef.bError,
					udiErrorID			=> stMcAxisOnline.stGetDriveRef.udiErrorID,
					stDriveRef			=> stMcAxisOnline.stDriveRef,
					Axis				:= Axis);
END_ACTION

ACTION ACT_Jog:
// Direct access from bSlow or bFast, if none then free choice
IF stMcAxisOnline.mcJog.bSlowForward OR stMcAxisOnline.mcJog.bSlowBackward THEN
	stMcAxisOnline.mcJog.eMode			:= MC_JOGMODE_STANDARD_SLOW;
ELSIF stMcAxisOnline.mcJog.bFastForward OR stMcAxisOnline.mcJog.bFastBackward THEN
	stMcAxisOnline.mcJog.eMode			:= MC_JOGMODE_STANDARD_FAST;
END_IF

mcJog(		Axis						:= Axis,
			JogForward					:= stMcAxisOnline.mcJog.bJogForward OR stMcAxisOnline.mcJog.bSlowForward OR stMcAxisOnline.mcJog.bFastForward,
			JogBackwards				:= stMcAxisOnline.mcJog.bJogBackwards OR stMcAxisOnline.mcJog.bSlowBackward OR stMcAxisOnline.mcJog.bFastBackward,
			Mode						:= stMcAxisOnline.mcJog.eMode,
			Position					:= stMcAxisOnline.mcJog.lrPosition,
			Velocity					:= stMcAxisOnline.mcJog.lrVelocity,
			Acceleration				:= stMcAxisOnline.mcJog.lrAcceleration,
			Deceleration				:= stMcAxisOnline.mcJog.lrDeceleration,
			Jerk						:= stMcAxisOnline.mcJog.lrJerk,
			Done						=> stMcAxisOnline.mcJog.bDone,
			Busy						=> stMcAxisOnline.mcJog.bBusy,
			Active						=> stMcAxisOnline.mcJog.bActive,
			CommandAborted				=> stMcAxisOnline.mcJog.bCommandAborted,
			Error						=> stMcAxisOnline.mcJog.bError,
			ErrorID						=> stMcAxisOnline.mcJog.udiErrorID);
END_ACTION

ACTION ACT_MotorMonitoring:
fbMotorMonitoring(	bReset				:= stMcAxisOnline.stMotorMonitoring.bReset,
					rTorqueLimit		:= stMcAxisOnline.stMotorMonitoring.rTorqueLimit,
					stDriveRef			:= stMcAxisOnline.stDriveRef,
					bError				=> stMcAxisOnline.stMotorMonitoring.bError,
					uiAdsErrId			=> stMcAxisOnline.stMotorMonitoring.uiAdsErrId,
					uiCANopenErrId		=> stMcAxisOnline.stMotorMonitoring.uiSecErrId,
					bInitialized		=> stMcAxisOnline.stMotorMonitoring.bInitialized,
					bWarning			=> stMcAxisOnline.stMotorMonitoring.bWarning,
					rWarningCurrent		=> stMcAxisOnline.stMotorMonitoring.rWarningCurrent,
					rTorquePerc			=> stMcAxisOnline.stMotorMonitoring.rTorquePerc,
					rTorquePercMax		=> stMcAxisOnline.stMotorMonitoring.rTorquePercMax,
					rTorque				=> stMcAxisOnline.stMotorMonitoring.rTorque,
					rTorqueF			=> stMcAxisOnline.stMotorMonitoring.rTorqueF,
					rTorqueMax			=> stMcAxisOnline.stMotorMonitoring.rTorqueMax,
					rCurrent			=> stMcAxisOnline.stMotorMonitoring.rCurrent,
					rCurrentF			=> stMcAxisOnline.stMotorMonitoring.rCurrentF,
					rCurrentMax			=> stMcAxisOnline.stMotorMonitoring.rCurrentMax,
					rI2T				=> stMcAxisOnline.stMotorMonitoring.rI2T,
					rI2TMax				=> stMcAxisOnline.stMotorMonitoring.rI2TMax,
					Axis				:= Axis);
END_ACTION

ACTION ACT_Move:
{region "Primary"}
mcMoveAbsolute(	Axis					:= Axis,
				Execute					:= stMcAxisOnline.mcMoveAbsolute.bExecute,
				Position				:= stMcAxisOnline.mcMoveAbsolute.lrPosition,
				Velocity				:= stMcAxisOnline.mcMoveAbsolute.lrVelocity,
				Acceleration			:= stMcAxisOnline.mcMoveAbsolute.lrAcceleration,
				Deceleration			:= stMcAxisOnline.mcMoveAbsolute.lrDeceleration,
				Jerk					:= stMcAxisOnline.mcMoveAbsolute.lrJerk,
				BufferMode				:= stMcAxisOnline.mcMoveAbsolute.eBufferMode,
				Options					:= stMcAxisOnline.mcMoveAbsolute.stOptions,
				Done					=> stMcAxisOnline.mcMoveAbsolute.bDone,
				Busy					=> stMcAxisOnline.mcMoveAbsolute.bBusy,
				Active					=> stMcAxisOnline.mcMoveAbsolute.bActive,
				CommandAborted			=> stMcAxisOnline.mcMoveAbsolute.bCommandAborted,
				Error					=> stMcAxisOnline.mcMoveAbsolute.bError,
				ErrorID					=> stMcAxisOnline.mcMoveAbsolute.udiErrorID);

mcMoveRelative(	Axis					:= Axis,
				Execute					:= stMcAxisOnline.mcMoveRelative.bExecute,
				Distance				:= stMcAxisOnline.mcMoveRelative.lrDistance,
				Velocity				:= stMcAxisOnline.mcMoveRelative.lrVelocity,
				Acceleration			:= stMcAxisOnline.mcMoveRelative.lrAcceleration,
				Deceleration			:= stMcAxisOnline.mcMoveRelative.lrDeceleration,
				Jerk					:= stMcAxisOnline.mcMoveRelative.lrJerk,
				BufferMode				:= stMcAxisOnline.mcMoveRelative.eBufferMode,
				Options					:= stMcAxisOnline.mcMoveRelative.stOptions,
				Done					=> stMcAxisOnline.mcMoveRelative.bDone,
				Busy					=> stMcAxisOnline.mcMoveRelative.bBusy,
				Active					=> stMcAxisOnline.mcMoveRelative.bActive,
				CommandAborted			=> stMcAxisOnline.mcMoveRelative.bCommandAborted,
				Error					=> stMcAxisOnline.mcMoveRelative.bError,
				ErrorID					=> stMcAxisOnline.mcMoveRelative.udiErrorID);
				
mcMoveVelocity(	Axis					:= Axis,
				Execute					:= stMcAxisOnline.mcMoveVelocity.bExecute,
				Velocity				:= stMcAxisOnline.mcMoveVelocity.lrVelocity,
				Acceleration			:= stMcAxisOnline.mcMoveVelocity.lrAcceleration,
				Deceleration			:= stMcAxisOnline.mcMoveVelocity.lrDeceleration,
				Jerk					:= stMcAxisOnline.mcMoveVelocity.lrJerk,
				Direction				:= stMcAxisOnline.mcMoveVelocity.eDirection,
				BufferMode				:= stMcAxisOnline.mcMoveVelocity.eBufferMode,
				Options					:= stMcAxisOnline.mcMoveVelocity.stOptions,
				InVelocity				=> stMcAxisOnline.mcMoveVelocity.bInVelocity,
				Busy					=> stMcAxisOnline.mcMoveVelocity.bBusy,
				Active					=> stMcAxisOnline.mcMoveVelocity.bActive,
				CommandAborted			=> stMcAxisOnline.mcMoveVelocity.bCommandAborted,
				Error					=> stMcAxisOnline.mcMoveVelocity.bError,
				ErrorID					=> stMcAxisOnline.mcMoveVelocity.udiErrorID);
stMcAxisOnline.mcMoveVelocity.bDone		:= stMcAxisOnline.mcMoveVelocity.bInVelocity;

mcMoveModulo(	Axis					:= Axis,
				Execute					:= stMcAxisOnline.mcMoveModulo.bExecute,
				Position				:= stMcAxisOnline.mcMoveModulo.lrPosition,
				Velocity				:= stMcAxisOnline.mcMoveModulo.lrVelocity,
				Acceleration			:= stMcAxisOnline.mcMoveModulo.lrAcceleration,
				Deceleration			:= stMcAxisOnline.mcMoveModulo.lrDeceleration,
				Jerk					:= stMcAxisOnline.mcMoveModulo.lrJerk,
				Direction				:= stMcAxisOnline.mcMoveModulo.eDirection,
				BufferMode				:= stMcAxisOnline.mcMoveModulo.eBufferMode,
				Options					:= stMcAxisOnline.mcMoveModulo.stOptions,
				Done					=> stMcAxisOnline.mcMoveModulo.bDone,
				Busy					=> stMcAxisOnline.mcMoveModulo.bBusy,
				Active					=> stMcAxisOnline.mcMoveModulo.bActive,
				CommandAborted			=> stMcAxisOnline.mcMoveModulo.bCommandAborted,
				Error					=> stMcAxisOnline.mcMoveModulo.bError,
				ErrorID					=> stMcAxisOnline.mcMoveModulo.udiErrorID);
{endregion}
{region "Secondary"}
mcMoveAbsolute2(Axis					:= Axis,
				Execute					:= stMcAxisOnline.mcMoveAbsolute2.bExecute,
				Position				:= stMcAxisOnline.mcMoveAbsolute2.lrPosition,
				Velocity				:= stMcAxisOnline.mcMoveAbsolute2.lrVelocity,
				Acceleration			:= stMcAxisOnline.mcMoveAbsolute2.lrAcceleration,
				Deceleration			:= stMcAxisOnline.mcMoveAbsolute2.lrDeceleration,
				Jerk					:= stMcAxisOnline.mcMoveAbsolute2.lrJerk,
				BufferMode				:= stMcAxisOnline.mcMoveAbsolute2.eBufferMode,
				Options					:= stMcAxisOnline.mcMoveAbsolute2.stOptions,
				Done					=> stMcAxisOnline.mcMoveAbsolute2.bDone,
				Busy					=> stMcAxisOnline.mcMoveAbsolute2.bBusy,
				Active					=> stMcAxisOnline.mcMoveAbsolute2.bActive,
				CommandAborted			=> stMcAxisOnline.mcMoveAbsolute2.bCommandAborted,
				Error					=> stMcAxisOnline.mcMoveAbsolute2.bError,
				ErrorID					=> stMcAxisOnline.mcMoveAbsolute2.udiErrorID);

mcMoveRelative2(Axis					:= Axis,
				Execute					:= stMcAxisOnline.mcMoveRelative2.bExecute,
				Distance				:= stMcAxisOnline.mcMoveRelative2.lrDistance,
				Velocity				:= stMcAxisOnline.mcMoveRelative2.lrVelocity,
				Acceleration			:= stMcAxisOnline.mcMoveRelative2.lrAcceleration,
				Deceleration			:= stMcAxisOnline.mcMoveRelative2.lrDeceleration,
				Jerk					:= stMcAxisOnline.mcMoveRelative2.lrJerk,
				BufferMode				:= stMcAxisOnline.mcMoveRelative2.eBufferMode,
				Options					:= stMcAxisOnline.mcMoveRelative2.stOptions,
				Done					=> stMcAxisOnline.mcMoveRelative2.bDone,
				Busy					=> stMcAxisOnline.mcMoveRelative2.bBusy,
				Active					=> stMcAxisOnline.mcMoveRelative2.bActive,
				CommandAborted			=> stMcAxisOnline.mcMoveRelative2.bCommandAborted,
				Error					=> stMcAxisOnline.mcMoveRelative2.bError,
				ErrorID					=> stMcAxisOnline.mcMoveRelative2.udiErrorID);
				
mcMoveVelocity2(Axis					:= Axis,
				Execute					:= stMcAxisOnline.mcMoveVelocity2.bExecute,
				Velocity				:= stMcAxisOnline.mcMoveVelocity2.lrVelocity,
				Acceleration			:= stMcAxisOnline.mcMoveVelocity2.lrAcceleration,
				Deceleration			:= stMcAxisOnline.mcMoveVelocity2.lrDeceleration,
				Jerk					:= stMcAxisOnline.mcMoveVelocity2.lrJerk,
				Direction				:= stMcAxisOnline.mcMoveVelocity2.eDirection,
				BufferMode				:= stMcAxisOnline.mcMoveVelocity2.eBufferMode,
				Options					:= stMcAxisOnline.mcMoveVelocity2.stOptions,
				InVelocity				=> stMcAxisOnline.mcMoveVelocity2.bInVelocity,
				Busy					=> stMcAxisOnline.mcMoveVelocity2.bBusy,
				Active					=> stMcAxisOnline.mcMoveVelocity2.bActive,
				CommandAborted			=> stMcAxisOnline.mcMoveVelocity2.bCommandAborted,
				Error					=> stMcAxisOnline.mcMoveVelocity2.bError,
				ErrorID					=> stMcAxisOnline.mcMoveVelocity2.udiErrorID);
stMcAxisOnline.mcMoveVelocity2.bDone	:= stMcAxisOnline.mcMoveVelocity2.bInVelocity;

mcMoveModulo2(	Axis					:= Axis,
				Execute					:= stMcAxisOnline.mcMoveModulo2.bExecute,
				Position				:= stMcAxisOnline.mcMoveModulo2.lrPosition,
				Velocity				:= stMcAxisOnline.mcMoveModulo2.lrVelocity,
				Acceleration			:= stMcAxisOnline.mcMoveModulo2.lrAcceleration,
				Deceleration			:= stMcAxisOnline.mcMoveModulo2.lrDeceleration,
				Jerk					:= stMcAxisOnline.mcMoveModulo2.lrJerk,
				Direction				:= stMcAxisOnline.mcMoveModulo2.eDirection,
				BufferMode				:= stMcAxisOnline.mcMoveModulo2.eBufferMode,
				Options					:= stMcAxisOnline.mcMoveModulo2.stOptions,
				Done					=> stMcAxisOnline.mcMoveModulo2.bDone,
				Busy					=> stMcAxisOnline.mcMoveModulo2.bBusy,
				Active					=> stMcAxisOnline.mcMoveModulo2.bActive,
				CommandAborted			=> stMcAxisOnline.mcMoveModulo2.bCommandAborted,
				Error					=> stMcAxisOnline.mcMoveModulo2.bError,
				ErrorID					=> stMcAxisOnline.mcMoveModulo2.udiErrorID);
{endregion}
END_ACTION

ACTION ACT_Power:
mcPower(	Axis						:= Axis,									//
			Enable						:= stMcAxisOnline.mcPower.bEnable,
			Enable_Positive				:= stMcAxisOnline.mcPower.bEnable_Positive,
			Enable_Negative				:= stMcAxisOnline.mcPower.bEnable_Negative,
			Override					:= stMcAxisOnline.mcPower.lrOverride,
			BufferMode					:= stMcAxisOnline.mcPower.eBufferMode,
			Options						:= stMcAxisOnline.mcPower.stOptions,
			Status						=> stMcAxisOnline.mcPower.bStatus,
			Busy						=> stMcAxisOnline.mcPower.bBusy,
			Active						=> stMcAxisOnline.mcPower.bActive,
			Error						=> stMcAxisOnline.mcPower.bError,
			ErrorID						=> stMcAxisOnline.mcPower.udiErrorID);
END_ACTION

ACTION ACT_Reset:
mcReset(	Axis						:= Axis,
			Execute						:= stMcAxisOnline.mcReset.bExecute,
			Done						=> stMcAxisOnline.mcReset.bDone,
			Busy						=> stMcAxisOnline.mcReset.bBusy,
			Error						=> stMcAxisOnline.mcReset.bError,
			ErrorID						=> stMcAxisOnline.mcReset.udiErrorID);
END_ACTION

ACTION ACT_SetPosition:
mcSetPosition(		Axis				:= Axis,
					Execute				:= stMcAxisOnline.mcSetPosition.bExecute,
					Position			:= stMcAxisOnline.mcSetPosition.lrPosition,
					Mode				:= stMcAxisOnline.mcSetPosition.bMode,
					Options				:= stMcAxisOnline.mcSetPosition.stOptions,
					Done				=> stMcAxisOnline.mcSetPosition.bDone,
					Busy				=> stMcAxisOnline.mcSetPosition.bBusy,
					Error				=> stMcAxisOnline.mcSetPosition.bError,
					ErrorID				=> stMcAxisOnline.mcSetPosition.udiErrorID);
END_ACTION

ACTION ACT_SetPositionIO:
fbSetPositionOffset(Execute				:= stMcAxisOnline.stSetPositionOffset.bExecute,
					Position			:= stMcAxisOnline.stSetPositionOffset.lrPosition,
					Relative			:= stMcAxisOnline.stSetPositionOffset.bRelative,
					Feedback			:= stMcAxisOnline.stSetPositionOffset.eFeedback,
					Memory				:= stMcAxisOnline.stSetPositionOffset.eMemory,
					Busy				=> stMcAxisOnline.stSetPositionOffset.bBusy,
					Error				=> stMcAxisOnline.stSetPositionOffset.bError,
					ErrorID				=> stMcAxisOnline.stSetPositionOffset.udiErrorID,
					Axis				:= Axis);
END_ACTION

ACTION ACT_States:
// Read States and forward main states
Axis.ReadStatus();
stMcAxisOnline.stStatus.stAxisStatus		:= Axis.Status;
stMcAxisOnline.stStatus.dwAxisId			:= Axis.NcToPlc.AxisId;
stMcAxisOnline.stStatus.bNcError			:= Axis.Status.Error;
stMcAxisOnline.stStatus.udiNcErrorCode		:= Axis.Status.ErrorID;
stMcAxisOnline.stStatus.udiNcErrorCodeHex	:= Axis.Status.ErrorID;

stMcAxisOnline.stStatus.sAxisName			:= stMcAxisOnline.stAxisParameter.sAxisName;
stMcAxisOnline.stStatus.lrActPos			:= Axis.NcToPlc.ActPos;
stMcAxisOnline.stStatus.lrModuloActPos		:= Axis.NcToPlc.ModuloActPos;
stMcAxisOnline.stStatus.lrActVelo			:= Axis.NcToPlc.ActVelo;
stMcAxisOnline.stStatus.lrActAcc			:= Axis.NcToPlc.ActAcc;
stMcAxisOnline.stStatus.lrActTorque			:= Axis.NcToPlc.ActTorque;
stMcAxisOnline.stStatus.lrPosDiff			:= Axis.NcToPlc.PosDiff;
stMcAxisOnline.stStatus.lrSetPos			:= Axis.NcToPlc.SetPos;
stMcAxisOnline.stStatus.lrSetVelo			:= Axis.NcToPlc.SetVelo;
stMcAxisOnline.stStatus.lrSetAcc			:= Axis.NcToPlc.SetAcc;
stMcAxisOnline.stStatus.lrSetTorque			:= Axis.NcToPlc.SetTorque;
stMcAxisOnline.stStatus.lrPosDiff			:= Axis.NcToPlc.PosDiff;
stMcAxisOnline.stStatus.bAxisReady			:= Axis.Status.Operational;
stMcAxisOnline.stStatus.bHomed				:= Axis.Status.Homed;
stMcAxisOnline.stStatus.bCoupled			:= Axis.Status.Coupled;

// zezwolenie na zjazd z krancowki hw
Axis.PlcToNc.ControlDWord.8				:= stMcAxisOnline.stStatus.bAcceptBlockedDrive;
END_ACTION

ACTION ACT_Stop:
mcHalt(		Axis						:= Axis,
			Execute						:= stMcAxisOnline.mcHalt.bExecute,
			Deceleration				:= stMcAxisOnline.mcHalt.lrDeceleration,
			Jerk						:= stMcAxisOnline.mcHalt.lrJerk,
			BufferMode					:= stMcAxisOnline.mcHalt.eBufferMode,
			Options						:= stMcAxisOnline.mcHalt.stOptions,
			Done						=> stMcAxisOnline.mcHalt.bDone,
			Busy						=> stMcAxisOnline.mcHalt.bBusy,
			Active						=> stMcAxisOnline.mcHalt.bActive,
			CommandAborted				=> stMcAxisOnline.mcHalt.bCommandAborted,
			Error						=> stMcAxisOnline.mcHalt.bError,
			ErrorID						=> stMcAxisOnline.mcHalt.udiErrorID);
			
mcStop(		Axis						:= Axis,
			Execute						:= stMcAxisOnline.mcStop.bExecute,
			Deceleration				:= stMcAxisOnline.mcStop.lrDeceleration,
			Jerk						:= stMcAxisOnline.mcStop.lrJerk,
			Options						:= stMcAxisOnline.mcStop.stOptions,
			Done						=> stMcAxisOnline.mcStop.bDone,
			Busy						=> stMcAxisOnline.mcStop.bBusy,
			Active						=> stMcAxisOnline.mcStop.bActive,
			CommandAborted				=> stMcAxisOnline.mcStop.bCommandAborted,
			Error						=> stMcAxisOnline.mcStop.bError,
			ErrorID						=> stMcAxisOnline.mcStop.udiErrorID);
			
mcStopSS2(	Axis						:= Axis,
			Execute						:= stMcAxisOnline.mcSS2.bExecute,
			Deceleration				:= stMcAxisOnline.mcSS2.lrDeceleration,
			Jerk						:= stMcAxisOnline.mcSS2.lrJerk,
			Options						:= stMcAxisOnline.mcSS2.stOptions,
			Done						=> stMcAxisOnline.mcSS2.bDone,
			Busy						=> stMcAxisOnline.mcSS2.bBusy,
			Active						=> stMcAxisOnline.mcSS2.bActive,
			CommandAborted				=> stMcAxisOnline.mcSS2.bCommandAborted,
			Error						=> stMcAxisOnline.mcSS2.bError,
			ErrorID						=> stMcAxisOnline.mcSS2.udiErrorID);
			
mcStopSS1(	Axis						:= Axis,
			Execute						:= stMcAxisOnline.mcSS1.bExecute,
			Deceleration				:= stMcAxisOnline.mcSS1.lrDeceleration,
			Jerk						:= stMcAxisOnline.mcSS1.lrJerk,
			Options						:= stMcAxisOnline.mcSS1.stOptions,
			Done						=> stMcAxisOnline.mcSS1.bDone,
			Busy						=> stMcAxisOnline.mcSS1.bBusy,
			Active						=> stMcAxisOnline.mcSS1.bActive,
			CommandAborted				=> stMcAxisOnline.mcSS1.bCommandAborted,
			Error						=> stMcAxisOnline.mcSS1.bError,
			ErrorID						=> stMcAxisOnline.mcSS1.udiErrorID);
// SS1 - after MC_Stop function we have to disable drive			
stMcAxisOnline.mcPower.bEnable R= stMcAxisOnline.mcPower.bEnable_Positive R= stMcAxisOnline.mcPower.bEnable_Negative R= (stMcAxisOnline.mcSS1.bDone OR stMcAxisOnline.mcSS1.bCommandAborted OR stMcAxisOnline.mcSS1.bError);
END_ACTION

ACTION ACT_SWLimitSwitch:
fbNcLimitSwitch(	udiAxisID		:= Axis.NcToPlc.AxisId, 
					bRead			:= stMcAxisOnline.stNcLimitSwitch.bRead, 
					bWrite			:= stMcAxisOnline.stNcLimitSwitch.bWrite, 
					bReset			:= stMcAxisOnline.stNcLimitSwitch.bReset, 
					lrSetMinPos		:= stMcAxisOnline.stNcLimitSwitch.lrSetMinPos, 
					lrSetMaxPos		:= stMcAxisOnline.stNcLimitSwitch.lrSetMaxPos, 
					bSetMinMon		:= stMcAxisOnline.stNcLimitSwitch.bSetMinMon, 
					bSetMaxMon		:= stMcAxisOnline.stNcLimitSwitch.bSetMaxMon, 
					bBusy			=> stMcAxisOnline.stNcLimitSwitch.bBusy, 
					bError			=> stMcAxisOnline.stNcLimitSwitch.bError, 
					udiErrorID		=> stMcAxisOnline.stNcLimitSwitch.udiErrorID, 
					lrActMinPos		=> stMcAxisOnline.stNcLimitSwitch.lrActMinPos, 
					lrActMaxPos		=> stMcAxisOnline.stNcLimitSwitch.lrActMaxPos, 
					bActMinMon		=> stMcAxisOnline.stNcLimitSwitch.bActMinMon, 
					bActMaxMon		=> stMcAxisOnline.stNcLimitSwitch.bActMaxMon);
END_ACTION

END_FUNCTION_BLOCK

// ---- POUs/FB/POUsAxisOnline/AX8000/FB_MotorMonitoringAX8000.TcPOU
//==================================================================================================
//							Beckhoff Automation Poland
//									4.07.2018
//	Blok funkcyjny pozwala na monitorowanie i ograniczanie momentu oraz monitoring parametru I2T dla AX8xxx.
//	Zmienne do zlinkowania zadeklarowane są wewnątrz bloku.
//	Ograniczenie i monitorowanie momentu
//	Ograniczenie momentu podawane jest przez wejście rTorqueLimit.
//	Na wyjściu podana jest wartość surowa w %, jak i przeskalowana na A (prąd) i Nm (moment).
//	Blok zwraca wartości bieżące, przefiltrowane i maksymalne.
//	Wartości maksymalne mogą być wyzerowane za pomocą zmiennej bReset.
//	Wewnętrznie wykorzystany jest blok FB_FilterEx.
//
//  v1.3	|| TC v 3.1.4022.22		|| - reset na poczatku bloku, optymalizacja kodu
//  v1.2	|| TC v 3.1.4022.16		|| - inicjalizacja po 10 nieudanych probach zglasza blad
//  v1.1	|| TC v 3.1.4022.16		|| - wyjscie iTorque przeniesione do lokalnych, w jego miejsce rTorquePerc i rTorquePercMax, 
//										flaga bTorqueLimitOK zalezna tylko od rTorqueLimitLow, zmiana nazw zgodnie z typami: uiAdsErrId, uiCANopenErrId
//  v1.0	|| TC v 3.1.4022.16		|| - pierwsza wersja
//==================================================================================================
FUNCTION_BLOCK FB_MotorMonitoringAX8000
VAR CONSTANT
	rTorqueLimitLow					: REAL 		:= 0.01;				// Low limit used for bipolar torque limit value
	rTorqueLimitHigh				: REAL		:= 500.0;				// High limit used for bipolar torque limit value
END_VAR
VAR_INPUT
	bReset							: BOOL;								// Reset FB
	rTorqueLimit					: REAL 		:= rTorqueLimitHigh; 	// Bipolar torque limit: 0-500%, resolution 0.1%, value goes to: 16#6072 (Ch A)/ 16#6872 (Ch B)
	stDriveRef						: ST_DriveRef;						// Necessary for FB_CoERead_ByDriveRef
END_VAR
VAR_OUTPUT
	bError							: BOOL; 							// General error: parameter or CoE read.
																		// If bError = TRUE and bInitialized = FALSE - error during read motor data.
																		// If bError = TRUE and bInitialized = TRUE and (iAdsErrId <> 0 or iCANopenErrId <> 0) then I2T read error
																		// If bError = TRUE and bInitialized = TRUE and iAdsErrId = 0 and iCANopenErrId = 0 then parameter error: rTorqueLimit outside permitted range rTorqueLimitLow..rTorqueLimitHigh or Empty stDriveRef
	uiAdsErrId						: UINT;								// Forwarded output FB_CoERead_ByDriveRef
	uiCANopenErrId					: UINT;								// Forwarded output FB_CoERead_ByDriveRef
	bInitialized					: BOOL;								// TRUE - Motor data read without errors, so it's possible to calculate torqe and current values in metric units
	bWarning						: BOOL;								// rCurrentF > rWarningCurrent, be aware to be over permitted range
	rWarningCurrent					: REAL; 							// Continuous Stall Current - motor parameter: 16#6075 (Ch A)/ 16#6875 (Ch B); scalled: [A]
	rTorquePerc						: REAL;								// [%]
	rTorquePercMax					: REAL;								// Max [%]
	rTorque							: REAL; 							// [Nm]
	rTorqueF						: REAL;								// Filtered [Nm]
	rTorqueMax						: REAL;								// Max [Nm]
	rCurrent						: REAL; 							// [A]
	rCurrentF						: REAL;								// Filtered [A]
	rCurrentMax						: REAL;								// Max [A]
	rI2T							: REAL; 							// Thermal Motor Utilization: 16#32C1:02 (Ch A)/ 16#36C1:02 (Ch B); units: [%]
	rI2TMax							: REAL; 							// Max % Nominal
END_VAR
VAR_IN_OUT
	Axis							: AXIS_REF;							// Axis Ref struct
END_VAR
VAR
//======================= Internal var ===========================
	iStep							: INT;								// Case instruction
	bDriveRefOK						: BOOL;								// stDriveRef contains necessary data to read CoE
	bTorqueLimitOK					: BOOL;								// rTorqueLimit in permitted range rTorqueLimitLow..rTorqueLimitHigh
	uiBipolarTorqueLimitValue  		AT %Q*: UINT; 						// Raw data, linked to Bipolar torque limit value
	iTorque 						: INT; 								// -1000 .. 1000 - RAW values the same as process image
	rTorqueRAW						: REAL; 							// -1000 .. 1000 - RAW values the same as process image
	rSfTorque						: REAL; 							// RAW -1000..1000 --> Nm
	rSfCurrent						: REAL; 							// Nm --> A
	udiMotorStandstillCurrent		: UDINT;							// 16#6075 (Ch A)/ 16#6875 (Ch B); units: [mA]
	udiMotorStandstillTorque		: UDINT;							// 16#6076 (Ch A)/ 16#6876 (Ch B); units: [mNm]
	wInitErrorCount					: WORD;								// Initialization error counter, if bigger then 10 then error
//========================== FBs ================================
	rtReset							: R_TRIG;							// Reset trigger
	tonWait							: TON;								// Wait timer - used for I2T read interval and for repeat initialization
	fbFilterEx						: FB_FilterEx;						// Filter
	fbCoERead						: FB_CoERead_ByDriveRef;			// FB for read CoE parameters
//===============================================================
END_VAR

//============== Reset max values and FB ========================
rtReset(CLK:= bReset);
IF rtReset.Q THEN
	fbCoERead.bExecute					:= FALSE;
	rCurrentMax							:= 0;
	rTorqueMax 							:= 0;
	rI2TMax								:= 0;
	uiAdsErrId		 					:= 0;
	uiCANopenErrId	 					:= 0;
	iStep								:= 0;
	wInitErrorCount						:= 0;
END_IF
//=================== Call triggers and timers ==================
tonWait(IN:= NOT tonWait.Q, PT:= T#1S);
//======= Check for parameter error - each cycle ================
bDriveRefOK 							:= (stDriveRef.nSlaveAddr <> 0) AND (stDriveRef.sNetId <> '');
bTorqueLimitOK 							:= (rTorqueLimit > rTorqueLimitLow);
//============= Read params and calculations ====================
CASE iStep OF
	
	0: // Read: Motor standstill current, 16#6075 (Ch A)/ 16#6875 (Ch B)
		// Execute read only if DriveRef is OK
		IF bDriveRefOK THEN
			fbCoERead.nIndex			:= 16#6075 + 16#800 * stDriveRef.nDriveNo;
			fbCoERead.nSubIndex			:= 0;
			fbCoERead.pDstBuf			:= ADR(udiMotorStandstillCurrent);
			fbCoERead.cbBufLen			:= SIZEOF(udiMotorStandstillCurrent);
			fbCoERead.bExecute			:= TRUE;
			iStep 						:= iStep + 10; 
		END_IF
	
	10: // Wait till read finish
		IF NOT fbCoERead.bBusy THEN
			IF fbCoERead.bError THEN
				fbCoERead.bExecute		:= FALSE;
				wInitErrorCount 		:= wInitErrorCount + 1;
				// Count > 10 then go to error and wait for reset, if not wait in warning step
				IF wInitErrorCount > 10 THEN
					uiAdsErrId			:= fbCoERead.iAdsErrId;
					uiCANopenErrId		:= fbCoERead.iCANopenErrId;
					iStep				:= 1000;									// Error step
				ELSE
					iStep				:= 900;										// Warning step
				END_IF
			ELSE
				fbCoERead.bExecute		:= FALSE;
				iStep 					:= iStep + 10;
			END_IF
		END_IF
	
	20: // Read: Motor standstill torque 16#6076 (Ch A)/ 16#6876 (Ch B)
		// Execute read only if DriveRef is OK
		IF bDriveRefOK THEN
			fbCoERead.nIndex			:= 16#6076 + 16#800 * stDriveRef.nDriveNo;
			fbCoERead.nSubIndex			:= 0;
			fbCoERead.pDstBuf			:= ADR(udiMotorStandstillTorque);
			fbCoERead.cbBufLen			:= SIZEOF(udiMotorStandstillTorque);
			fbCoERead.bExecute			:= TRUE;
			iStep 						:= iStep + 10; 
		END_IF
	
	30:	// Wait till read finish
		IF NOT fbCoERead.bBusy THEN
			IF fbCoERead.bError THEN
				fbCoERead.bExecute		:= FALSE;
				wInitErrorCount 		:= wInitErrorCount + 1;
				// Count > 10 then go to error and wait for reset, if not wait in warning step
				IF wInitErrorCount > 10 THEN
					uiAdsErrId			:= fbCoERead.iAdsErrId;
					uiCANopenErrId		:= fbCoERead.iCANopenErrId;
					iStep				:= 1000;									// Error step
				ELSE
					iStep				:= 900;										// Warning step
				END_IF
			ELSE
				fbCoERead.bExecute		:= FALSE;
				iStep 					:= iStep + 10;
			END_IF
		END_IF
	
	40: // Calculate Sf
		rSfTorque						:= UDINT_TO_REAL(udiMotorStandstillTorque) / 1000000;
		rSfCurrent						:= UDINT_TO_REAL(udiMotorStandstillCurrent) / 1000000;
		rWarningCurrent					:= UDINT_TO_REAL(udiMotorStandstillCurrent) / 1000;
		iStep 							:= 100;
	
	100: // Read: Thermal Motor Utilization (I2T), 16#32C1:02 (Ch A)/ 16#36C1:02 (Ch B)
		fbCoERead.nIndex				:= 16#32C1 + (16#400 * stDriveRef.nDriveNo);
		fbCoERead.nSubIndex				:= 02;
		fbCoERead.pDstBuf				:= ADR(rI2T);
		fbCoERead.cbBufLen				:= SIZEOF(rI2T);
		fbCoERead.bExecute				:= bDriveRefOK AND tonWait.Q;				// Execute read only if DriveRef is OK
		IF fbCoERead.bBusy THEN
			iStep 						:= iStep + 10;
		END_IF
	
	110: // Wait till read finish
		IF NOT fbCoERead.bBusy THEN
			IF fbCoERead.bError OR NOT bTorqueLimitOK OR NOT bDriveRefOK THEN
				uiAdsErrId				:= fbCoERead.iAdsErrId;
				uiCANopenErrId			:= fbCoERead.iCANopenErrId;
				iStep					:= 1000;									// Error step
			ELSE
				iStep 					:= iStep - 10;				
			END_IF
		END_IF
	
	900: // Warning - wait and repeat read - problem during read motor data, i.e. EtherCAT doesn't work yet
		IF tonWait.Q THEN
			iStep 						:= 0;	// Repeat initialization phase 
		END_IF
			  
			  
	1000: // Error - wait for reset 
		;
END_CASE
//===============================================================
	 
bError			 						:= iStep = 1000;
bInitialized	 						:= iStep >= 100 AND NOT bError;
//====================== Call CoE read FB =======================
fbCoERead(stDriveRef:= stDriveRef);
//======================== Set outputs ==========================
rTorquePerc								:= LREAL_TO_REAL(Axis.NcToPlc.ActTorque); 		// [%]
rTorqueRAW 								:= rTorquePerc*10;								// -1000 .. 1000 - RAW values the same as process image
//===================== Filter current value ====================
fbFilterEx(rIn:= rTorqueRAW, tTimeConstant:= T#1S);

iTorque 								:= REAL_TO_INT(rTorqueRAW);
rTorque 								:= rTorqueRAW * rSfTorque;
rCurrent 								:= rTorqueRAW * rSfCurrent;
rTorqueF 								:= fbFilterEx.rOut * rSfTorque;
rCurrentF 								:= fbFilterEx.rOut * rSfCurrent;
//=============== Save torque and current max values ===============
IF ABS(rCurrentMax) < ABS(rCurrentF) THEN
	rTorquePercMax						:= rTorquePerc;
	rCurrentMax 						:= rCurrentF;
	rTorqueMax 							:= rTorqueF;
END_IF
//======================== Save I2T max value ======================
IF rI2TMax < rI2T THEN
	rI2TMax 							:= rI2T;
END_IF

//===================== Limit output torque =====================
IF rTorqueLimit < rTorqueLimitLow THEN
	uiBipolarTorqueLimitValue 			:= REAL_TO_UINT(rTorqueLimitHigh);			// Secure against 0 value - probably empty var connected to input
ELSE
	uiBipolarTorqueLimitValue 			:= REAL_TO_UINT(LIMIT(rTorqueLimitLow,rTorqueLimit,rTorqueLimitHigh))*10;
END_IF
//========================= Warning =============================
bWarning								:= rCurrentF > rWarningCurrent;

END_FUNCTION_BLOCK

// ---- POUs/FB/POUsAxisOnline/AX8000/FB_HoldingBrakeCtrlAX8000.TcPOU
//==================================================================================================
//							Beckhoff Automation Poland
//									12.04.2018
//	Blok funkcyjny kontroli luzownika w silniku podpietym do AX8000. Przewaga ForceLock
//	Dzialania na obiekcie: 3000:07 Motor brake force
//	Index:			AxisMainSlot: 16#3000 (Ch A)/ 16#3400 (Ch B)
//	Subindex:		16#07
//	Datatype:		ENUM (INT16)
//	Enum Value:		0 (0x00): 	Release_force
//					1 (0x01): 	Force_lock
//					2 (0x02): 	Force_unlock
//
//  v1.0	|| TC v 3.1.4022.16		|| - pierwsza wersja
//==================================================================================================
FUNCTION_BLOCK FB_HoldingBrakeCtrlAX8000
VAR_INPUT
	bForceLock 						: BOOL;								// 
	bForceUnlock					: BOOL;								// 
	stDriveRef						: ST_DriveRef;
END_VAR
VAR_OUTPUT
	bBusy							: BOOL;
	bError							: BOOL; 							// General error: parameter or CoE read.
																		// If bError = TRUE and bInitialized = FALSE - error during read motor data.
																		// If bError = TRUE and bInitialized = TRUE and (iAdsErrId <> 0 or iCANopenErrId <> 0) then I2T read error
																		// If bError = TRUE and bInitialized = TRUE and iAdsErrId = 0 and iCANopenErrId = 0 then parameter error: rTorqueLimit outside permitted range rTorqueLimitLow..rTorqueLimitHigh or Empty stDriveRef
	iAdsErrId						: UINT;								// Forwarded output FB_CoERead_ByDriveRef
	iCANopenErrId					: UINT;								// Forwarded output FB_CoERead_ByDriveRef
END_VAR
VAR
	bExecute						: BOOL;
	iMotorBrakeForce				: INT;								// 0 - Release_force, 1 - Force_lock, 2 - Force_unlock
	rtForceLock						: R_TRIG;
	rtForceUnlock					: R_TRIG;
	ftForceLock						: F_TRIG;
	ftForceUnlock					: F_TRIG;
	fbForceLockUnlock				: FB_CoEWrite_ByDriveRef;
END_VAR

{region "Call triggers"}
//======================= Call triggers =========================
rtForceLock(CLK:= bForceLock);
ftForceLock(CLK:= bForceLock);
rtForceUnlock(CLK:= bForceUnlock);
ftForceUnlock(CLK:= bForceUnlock);
bExecute								:= rtForceLock.Q OR ftForceLock.Q OR rtForceUnlock.Q OR ftForceUnlock.Q;
//===============================================================
{endregion}
{region "Main code"}
//========================= Main code ===========================
IF bExecute THEN
	iMotorBrakeForce 						:= 0;										// Clear value
	iMotorBrakeForce.1 						:= bForceUnlock;							// Set force unlock bit
	iMotorBrakeForce 						:= SEL(bForceLock, iMotorBrakeForce, 1);	// Set force lock bit, it has higher priority than unlock
END_IF

fbForceLockUnlock(	stDriveRef				:= stDriveRef, 
					nIndex					:= 16#3000 + (stDriveRef.nDriveNo * 16#400), 
					nSubIndex				:= 16#07, 
					pSrcBuf					:= ADR(iMotorBrakeForce), 
					cbBufLen				:= SIZEOF(iMotorBrakeForce), 
					bExecute				:= bExecute,
					bBusy					=> bBusy, 
					bError					=> bError, 
					iAdsErrId				=> iAdsErrId, 
					iCANopenErrId			=> iCANopenErrId);
//===============================================================
{endregion}

END_FUNCTION_BLOCK

// ---- POUs/FB/POUsAxisOnline/AX8000/FB_ReadChannelErrorCodeAX8000.TcPOU
//==================================================================================================
//							Beckhoff Automation Poland
//									11.04.2018
//	This object shall provide the text id of the last DiagMessage of type error, which occurred in this axis.
//  v1.0	|| TC v 3.1.4022.16		|| - pierwsza wersja
//==================================================================================================
FUNCTION_BLOCK FB_ReadChannelErrorCodeAX8000
VAR_INPUT
	bExecute 						: BOOL;
	stDriveRef						: ST_DriveRef;						// 
END_VAR
VAR_OUTPUT
	bBusy							: BOOL;
	bError							: BOOL; 							// General error: parameter or CoE read.
	iAdsErrId						: UINT;								// Forwarded output FB_CoERead_ByDriveRef
	iCANopenErrId					: UINT;								// Forwarded output FB_CoERead_ByDriveRef
	uiChannelErrorCode				: UINT;								// 603F Error code	0x603F (Ch A)/ 0x683F (Ch B) 	UINT16
	{attribute 'displaymode':='hex'}
	uiChannelErrorCodeHex			: UINT;								// 603F Error code	0x603F (Ch A)/ 0x683F (Ch B) 	UINT16
END_VAR
VAR
	fbCoERead						: FB_CoERead_ByDriveRef;			// FB for read CoE parameters
END_VAR

fbCoERead(	stDriveRef					:= stDriveRef,
			nIndex						:= 16#603F + (stDriveRef.nDriveNo * 16#800),
			nSubIndex					:= 0,
			pDstBuf						:= ADR(uiChannelErrorCode),
			cbBufLen					:= SIZEOF(uiChannelErrorCode),
			bExecute					:= bExecute,
			bBusy						=> bBusy,
			bError						=> bError,
			iAdsErrId					=> iAdsErrId,
			iCANopenErrId				=> iCANopenErrId);

uiChannelErrorCodeHex					:= uiChannelErrorCode;

END_FUNCTION_BLOCK

// ---- POUs/FB/POUsAxisOnline/FBs/FB_GetDriveRef.TcPOU
//==================================================================================================
//							Beckhoff Automation Poland
//									28.03.2018
//	Blok funkcyjny tworzacy strukture ST_DriveRef z AXIS_REF
//	Przydatny w komunikacji CoE w AX8000
//  v1.0	|| TC v 3.1.4022.16		|| - pierwsza wersja
//==================================================================================================
FUNCTION_BLOCK FB_GetDriveRef
VAR_INPUT
	bExecute								: BOOL;							// rising edge starts sequence
END_VAR
VAR_OUTPUT
	bBusy									: BOOL;
	bError									: BOOL;	
	udiErrorID								: UDINT;						// bError=TRUE AND udiErrorID=0 means state request timeout
	stDriveRef								: ST_DriveRef;					// come from stPlcDriveRef
END_VAR
VAR_IN_OUT
	Axis									: AXIS_REF;
END_VAR
VAR
	fbAdsRead								: ADSREAD;
	ftADSRead								: F_TRIG;
	stPlcDriveRef							: ST_PlcDriveRef;				// ADS buffer (need to change aNetId into sNetId)
END_VAR
VAR CONSTANT
	NCIDXG_AXPARMS							: UDINT			:= 16#4000;		// ADS group number to axis parameters 
	NCIDXO_AXP_HWAMSADDR					: UDINT			:= 16#31;		// ADS offset to drive channel
END_VAR

fbAdsRead(	NETID			:= '', 
			PORT			:= AMSPORT_R0_NC, 								// set ADS Port to NC
			IDXGRP			:= NCIDXG_AXPARMS + Axis.NcToPlc.AxisId,		// set ADS Group to AXIS Parameters 
			IDXOFFS			:= NCIDXO_AXP_HWAMSADDR,						// set ADS offset to channel number 
			LEN				:= SIZEOF(stPlcDriveRef), 
			DESTADDR		:= ADR(stPlcDriveRef), 
			READ			:= bExecute, 
			BUSY			=> bBusy, 
			ERR				=> bError, 
			ERRID			=> udiErrorID);
			
ftADSRead(CLK:= bBusy);

IF ftADSRead.Q AND NOT fbAdsRead.ERR THEN	
	stDriveRef.sNetId		:= F_CreateAmsNetId(stPlcDriveRef.aNetId);		// change AmsNetId array into string
	stDriveRef.nSlaveAddr	:= stPlcDriveRef.nSlaveAddr;
	stDriveRef.nDriveNo		:= stPlcDriveRef.nDriveNo;			
END_IF

END_FUNCTION_BLOCK

// ---- POUs/FB/Axis/F_AX8xErrMsg.TcPOU
//==================================================================================================
//							Beckhoff Automation Poland
//								7.12.2018
//		Funkcja konwertujaca nr bledu na opis
// 	v1.0	|| TC v 3.1.4022.27	|| - pierwsza wersja
//==================================================================================================
FUNCTION F_AX8xErrMsg : STRING(255)
VAR_INPUT
	uiDriveError : UINT;
END_VAR

IF uiDriveError < 1 THEN
	F_AX8xErrMsg := '';
	RETURN;
END_IF

CASE uiDriveError OF
	16#2220: F_AX8xErrMsg:= '2220 =  Continuous over current (device internal)';
	16#2310: F_AX8xErrMsg:= '2310 =  Continuous over current (device output side)';
	16#2330: F_AX8xErrMsg:= '2330 = Earth leakage (motor-side)';
	16#2340: F_AX8xErrMsg:= '2340 =  Short circuit (motor-side)';
	16#2380: F_AX8xErrMsg:= '2380 =  Continuous over current (device output side) Phase U';
	16#2381: F_AX8xErrMsg:= '2381 =  Continuous over current (device output side) Phase V';
	16#2382: F_AX8xErrMsg:= '2382 =  Continuous over current (device output side) Phase W';
	16#2383: F_AX8xErrMsg:= '2383 =  Phase U current offset out of range';
	16#2384: F_AX8xErrMsg:= '2384 =  Phase V current offset out of range';
	16#2385: F_AX8xErrMsg:= '2385 =  Phase W current offset out of range';
	16#3110: F_AX8xErrMsg:= '3110 =  Mains over-voltage';
	16#3120: F_AX8xErrMsg:= '3120 =  Mains under-voltage';
	16#3130: F_AX8xErrMsg:= '3130 =  Phase failure';
	16#3180: F_AX8xErrMsg:= '3180 =  Phase failure motor or Mains voltage over brake resistor operating voltage';
	16#3181: F_AX8xErrMsg:= '3181 =  Phase frequency (motor-side) raised above 600 Hz or Wrong mains type';
	16#3182: F_AX8xErrMsg:= '3182 =  Velocity actual Value raised above the max channel accepted velocity';
	16#3183: F_AX8xErrMsg:= '3183 = The bipolar velocity limit is higher than 1/4 of position range limit per EtherCAT Sync1 cycle.';
	16#3210: F_AX8xErrMsg:= '3210 =  DC link over-voltage';
	16#3220: F_AX8xErrMsg:= '3220 =  DC link undervoltage';
	16#3280: F_AX8xErrMsg:= '3280 =  DC link is not ready or  Device DC link over-voltage';
	16#4110: F_AX8xErrMsg:= '4110 =  Excess ambient temperature';
	16#4210: F_AX8xErrMsg:= '4210 =  Excess temperature device';
	16#4310: F_AX8xErrMsg:= '4310 =  Drive overtemperature shut down';
	16#4380: F_AX8xErrMsg:= '4380 =  Fan speed seems to be zero.';
	16#5112: F_AX8xErrMsg:= '5112 =  Supply low voltage: supply +24V';
	16#5180: F_AX8xErrMsg:= '5180 =  Output stage STO active.';
	16#5181: F_AX8xErrMsg:= '5181 =  Power supply status,  torque off order';
	16#5182: F_AX8xErrMsg:= '5182 =  Power supply status inactive';
	16#5183: F_AX8xErrMsg:= '5183 =  Power supply status,  NC handling order';
	16#5184: F_AX8xErrMsg:= '5184 =  Supply DC-link circuit is not ready';
	16#5185: F_AX8xErrMsg:= '5185 =  Power supply status,  non-regenerative brake order';
	16#5186: F_AX8xErrMsg:= '5186 =  Power supply status,  regenerative brake order';
	16#5187: F_AX8xErrMsg:= '5187 =  Power supply communication is not established';
	16#5190: F_AX8xErrMsg:= '5190 =  Test 5V supply failed';
	16#5192: F_AX8xErrMsg:= '5192 =  Supply high voltage: supply +24V';
	16#5441: F_AX8xErrMsg:= '5441 =  Positive limit switch active';
	16#5442: F_AX8xErrMsg:= '5442 =  Negative limit switch active';
	16#5580: F_AX8xErrMsg:= '5580 =  Read failure EEPROM';
	16#5581: F_AX8xErrMsg:= '5581 =  Checksum failure EEPROM';
	16#5582: F_AX8xErrMsg:= '5582 =  EEPROM contains blank Data';
	16#5583: F_AX8xErrMsg:= '5583 =  Unexpected EEPROM';
	16#5584: F_AX8xErrMsg:= '5584 =  EEPROM contains blank Data';
	16#5585: F_AX8xErrMsg:= '5585 =  Unexpected EEPROM';
	16#5586: F_AX8xErrMsg:= '5586 =  Restored Errormessages from persistant memory';
	16#5587: F_AX8xErrMsg:= '5587 =  Missing factory settings in eeprom';
	16#5588: F_AX8xErrMsg:= '5588 =  Missing ids in eeprom display board';
	16#5589: F_AX8xErrMsg:= '5589 =  Read failure eeprom display board';
	16#5590: F_AX8xErrMsg:= '5590 =  Detected incompatible Pcb';
	16#5591: F_AX8xErrMsg:= '5591 =  Identity incompatible to a Pcb';
	16#5592: F_AX8xErrMsg:= '5592 =  FirmwareIndex is incompatible to this Firmware.';
	16#5593: F_AX8xErrMsg:= '5593 =  Structure Version is incompatible to this Firmware';
	16#5594: F_AX8xErrMsg:= '5594 =  Simulating persistent data features.';
	16#5595: F_AX8xErrMsg:= '5595 =  Modulo remainder will not be stored.';
	16#5596: F_AX8xErrMsg:= '5596 =  Storing of persistant data failed.';
	16#6010: F_AX8xErrMsg:= '6010 =  Software reset (watchdog)';
	16#6080: F_AX8xErrMsg:= '6080 =  Failure config bits';
	16#6180: F_AX8xErrMsg:= '6180 =  Internal Software Error Type A';
	16#6181: F_AX8xErrMsg:= '6181 =  Internal Software Error Type B';
	16#6182: F_AX8xErrMsg:= '6182 =  Internal Software Error Type C';
	16#6183: F_AX8xErrMsg:= '6183 =  Internal Watchdog Error';
	16#6190: F_AX8xErrMsg:= '6190 =  Init Timeout';
	16#6310: F_AX8xErrMsg:= '6310 =  Loss of parameters';
	16#6320: F_AX8xErrMsg:= '6320 =  Parameter error';
	16#6380: F_AX8xErrMsg:= '6380 =  Parameter Interpolator: Illegal Interpolation sub mode select or  Parameters x with parametrized y is too low.';
	16#6381: F_AX8xErrMsg:= '6381 =  Parameter x with parametrized y is too high';
	16#6382: F_AX8xErrMsg:= '6382 =  Illegal Slotconfiguration. Slot is empty.';
	16#6383: F_AX8xErrMsg:= '6383 =  Illegal Slotconfiguration. Double Feedback Selection.';
	16#6384: F_AX8xErrMsg:= '6384 =  Illegal Slotconfiguration. Slot has to be empty.';
	16#6385: F_AX8xErrMsg:= '6385 =  Parameter Interpolator. Operation Mode does not match';
	16#6386: F_AX8xErrMsg:= '6386 =  Parameter Interpolator: Illegal NC-Task cycle time';
	16#6387: F_AX8xErrMsg:= '6387 =  Parameter Motor. The configured DCLink Max Voltage is higher than the Motor Max Voltage.';
	16#6388: F_AX8xErrMsg:= '6388 =  Parameter Torque Control: The value in Object 0x%x/%x is higher than the Motor peak current (0x%x/%x).';
	16#6389: F_AX8xErrMsg:= '6389 =  Parameter Torque Control: The value in Object 0x%x/%x is higher than the Configured peak current (0x%x/%x).';
	16#6390: F_AX8xErrMsg:= '6390 =  Factor Group Parameters: Feed constant illegal feed';
	16#6391: F_AX8xErrMsg:= '6391 =  Factor Group Parameters: Feed constant illegal shaft revolutions';
	16#6392: F_AX8xErrMsg:= '6392 =  Factor Group Parameters: Gear ratio illegal Motor shaft revolutions';
	16#6393: F_AX8xErrMsg:= '6393 =  Factor Group Parameters: Gear ratio illegal Driving shaft revolutions';
	16#6394: F_AX8xErrMsg:= '6394 =  Factor Group Parameters: Position encoder resolution illegal encoder increments';
	16#6395: F_AX8xErrMsg:= '6395 =  Factor Group Parameters: Position encoder resolution illegal motor revolutions';
	16#6396: F_AX8xErrMsg:= '6396 =  additional Factor Group Parameters: Feed constant illegal feed';
	16#6397: F_AX8xErrMsg:= '6397 =  additional Factor Group Parameters: Feed constant illegal shaft revolutions';
	16#6398: F_AX8xErrMsg:= '6398 =  additional Factor Group Parameters: Gear ratio illegal Motor shaft revolutions';
	16#6399: F_AX8xErrMsg:= '6399 =  additional Factor Group Parameters: Gear ratio illegal Driving shaft revolutions';
	16#7111: F_AX8xErrMsg:= '7111 =  Failure brake chopper';
	16#7112: F_AX8xErrMsg:= '7112 =  Over current brake chopper';
	16#7122: F_AX8xErrMsg:= '7122 =  Motor error or commutation malfunction';
	16#7180: F_AX8xErrMsg:= '7180 =  Motor brake: Current monitoring error. Or  Brake resistor not found';
	16#7181: F_AX8xErrMsg:= '7181 =  Motor thermal utilization has reached the warning level.  Or  Brake resistor power overload by DC link over-voltage';
	16#7182: F_AX8xErrMsg:= '7182 =  Motor thermal utilization has left the warning level. Or  Wrong xml file';
	16#7183: F_AX8xErrMsg:= '7183 =  Motor thermal utilization has reached the Error Level';
	16#7184: F_AX8xErrMsg:= '7184 =  Motor overload shut down';
	16#7185: F_AX8xErrMsg:= '7185 =  Motor overtemperature shut down';
	16#7186: F_AX8xErrMsg:= '7186 = Detected moving axis on enable transition.';
	16#7320: F_AX8xErrMsg:= '7320 =  HpfDsl: Encoder error (position invalid)';
	16#7380: F_AX8xErrMsg:= '7380 =  Current sensor motor phase U or HpfDsl: Encoder start sequence failed';
	16#7381: F_AX8xErrMsg:= '7381 =  Current sensor motor phase V or HpfDsl: Encoder shutdown failed';
	16#7382: F_AX8xErrMsg:= '7382 =  Current sensor motor phase W or HpfDsl: Parameter access error';
	16#7383: F_AX8xErrMsg:= '7383 =  HpfDsl: Internal error';
	16#7384: F_AX8xErrMsg:= '7384 =  HpfDsl: Cyclic monitoring error';
	16#7385: F_AX8xErrMsg:= '7385 =  HpfDsl: Encoder file processing';
	16#7386: F_AX8xErrMsg:= '7386 =  HpfDsl: Found no encoder (No link to an encoder)!';
	16#7580: F_AX8xErrMsg:= '7580 =  I2C_communication_failure';
	16#8180: F_AX8xErrMsg:= '8180 =  System restart or sync lost';
	16#8181: F_AX8xErrMsg:= '8181 =  Lost Distributed clocks Sync';
	16#8182: F_AX8xErrMsg:= '8182 =  EtherCAT Statemachine shutdown with enabled Axis';
	16#8183: F_AX8xErrMsg:= '8183 =  Controlword output cycle counter monitoring';
	16#8480: F_AX8xErrMsg:= '8480 = Overspeed error';
	16#8611: F_AX8xErrMsg:= '8611 = Following error';
	16#8680: F_AX8xErrMsg:= '8680 =  Position Demand Value outside of the specified Position Range Limits';
	16#8780: F_AX8xErrMsg:= '8780 =  Configured Sync1 Cycle Time is above Maximum';
	16#8781: F_AX8xErrMsg:= '8781 =  Configured Sync1 Cycle Time is below Minimum';
	16#8782: F_AX8xErrMsg:= '8782 =  Configured Sync1 Cycle Time is not a multiple of the Sync0 Cycle Time';
	16#8783: F_AX8xErrMsg:= '8783 =  Configured Sync0 Cycle Time is not legal';
	16#638A: F_AX8xErrMsg:= '638A =  The Axis seems not to be parameterised.';
	16#638B: F_AX8xErrMsg:= '638B =  Parameter Torque Current curve: Unable to calculate Torque Current curve.';
	16#638C: F_AX8xErrMsg:= '638C =  Motor type does not match';
	16#638D: F_AX8xErrMsg:= '638D =  Connected Motor is compatible to the configured Motor';
	16#638E: F_AX8xErrMsg:= '638E =  The Motor brake is automatically unlocked';
	16#638F: F_AX8xErrMsg:= '638F =  Parameter Torque Control: The value in Object 0x%x/%x is higher then the Motor maximum voltage slope (0x%x/%x).';
	16#639A: F_AX8xErrMsg:= '639A =  additional Factor Group Parameters: Position encoder resolution illegal encoder increments';
	16#639B: F_AX8xErrMsg:= '639B =  additional Factor Group Parameters: Position encoder resolution illegal motor revolutions';
	16#639C: F_AX8xErrMsg:= '639C =  Velocity factor illegal. A possible Value would be %u/%u.';
	16#639D: F_AX8xErrMsg:= '639D =  Acceleration factor illegal. A possible Value would be %u/%u.';
	16#639E: F_AX8xErrMsg:= '639E =  Scaling index object 0x%x does not fit the Factor group parameters for the first Encoder';
	16#639F: F_AX8xErrMsg:= '639F =  Scaling index object 0x%x does not fit the Factor group parameters for the second Encoder';
	16#63A0: F_AX8xErrMsg:= '63A0 =  Motor or Primary Feedback changed';
	16#63A1: F_AX8xErrMsg:= '63A1 =  Secondary Feedback changed';
	16#63A2: F_AX8xErrMsg:= '63A2 =  Offset position actual value: No position offset existing in source "encoder memory"';
	16#63A3: F_AX8xErrMsg:= '63A3 =  Offset additional position actual value: No position offset existing in source "encoder memory"';
	16#63A4: F_AX8xErrMsg:= '63A4 =  Offset position actual value: No position offset existing in source "drive memory"';
	16#63A5: F_AX8xErrMsg:= '63A5 =  Offset additional position actual value: No position offset existing in source "drive memory"';
	16#63A6: F_AX8xErrMsg:= '63A6 =  Jerk factor illegal. A possible Value would be %u/%u.';
	16#63A7: F_AX8xErrMsg:= '63A7 =  The range %u of the Position range limit is below the minimum accepted value of %u.';
	16#63A8: F_AX8xErrMsg:= '63A8 =  Position range limit Inc with remainder is not supported for primary feedback.';
	16#63A9: F_AX8xErrMsg:= '63A9 =  Position range limit Inc with remainder is not supported for secondary feedback.';
	16#63AA: F_AX8xErrMsg:= '63AA =  Object 0x%X/%X changed in EtherCAT SafeOP or OP.';
	16#8A80: F_AX8xErrMsg:= '8A80 =  Illegal Modes of Operation';
	16#8A81: F_AX8xErrMsg:= '8A81 =  Illegal Modes of Operation change';
	16#A000: F_AX8xErrMsg:= 'A000 =  Transition Pre-Op to Safe-Op not successful. Sync Manager Length Error.';
	16#A001: F_AX8xErrMsg:= 'A001 =  Transition Pre-Op to Safe-Op not successful. Sync Manager Address Error.';
	16#A002: F_AX8xErrMsg:= 'A002 =  Transition Pre-Op to Safe-Op not successful. Sync Manager Settings Error.';
	16#A003: F_AX8xErrMsg:= 'A003 =  Transition Pre-Op to Safe-Op not successful. Sync Manager Address Range overlap.';
	16#A004: F_AX8xErrMsg:= 'A004 =  Sync Manager is disabledand has a Size unequal zero.';
	16#A010: F_AX8xErrMsg:= 'A010 =  SDO Complete Access Error: Object 0x%x/%x';
	16#A011: F_AX8xErrMsg:= 'A011 =  RxPdo Mapping Error: Unable to map Object (not possible).';
	16#A012: F_AX8xErrMsg:= 'A012 =  TxPdo Mapping Error: Unable to map Object (not possible).';
	16#A013: F_AX8xErrMsg:= 'A013 =  RxPdo Mapping Error: Double Mapping of Object.';
	16#A014: F_AX8xErrMsg:= 'A014 =  TxPdo Mapping Error: Double Mapping of Object.';
	16#A015: F_AX8xErrMsg:= 'A015 =  RxPdo Mapping Error: Unable to map Object (no Mappings left).';
	16#A016: F_AX8xErrMsg:= 'A016 =  TxPdo Mapping Error: Unable to map Object (no Mappings left).';
	16#A017: F_AX8xErrMsg:= 'A017 =  RxPdo Mapping Error: Object always has to be mapped.';
	16#A018: F_AX8xErrMsg:= 'A018 =  TxPdo Mapping Error: Object 0x%x/%x always has to be mapped.';
	16#A019: F_AX8xErrMsg:= 'A019 =  RxPdo Mapping Error: Object has to be mapped because of modes of operation.';
	16#A01A: F_AX8xErrMsg:= 'A01A =  TxPdo Mapping Error: Object has to be mapped because of modes of operation.';
	16#A01B: F_AX8xErrMsg:= 'A01B =  RxPdo BitMapping Error: Object 0x%x/%x is not next to Object 0x%x/%x. (SyncManager %u)';
	16#A01C: F_AX8xErrMsg:= 'A01C =  TxPdo BitMapping Error: Object 0x%x/%x is not next to Object 0x%x/%x. (SyncManager %u)';
	16#A01D: F_AX8xErrMsg:= 'A01D =  RxPdo BitMapping Error: Can not Transform Bit-Mappings to Byte-Mappings. (SyncManager %u)';
	16#A01E: F_AX8xErrMsg:= 'A01E =  TxPdo BitMapping Error: Can not Transform Bit-Mappings to Byte-Mappings. (SyncManager %u)';
	16#A080: F_AX8xErrMsg:= 'A080 =  Safe-Op is not possible because the local TwinCAT Runtime is in ConfigMode.';
	16#A081: F_AX8xErrMsg:= 'A081 =  Transition Pre-Op to Safe-Op not successful. Safetycard not detected.';
	16#A082: F_AX8xErrMsg:= 'A082 =  EtherCAT Slave Stack Error:';
	16#FF01: F_AX8xErrMsg:= 'FF01 =  Init Timeout or Error reaction forced: Generative brake order';
	16#FF02: F_AX8xErrMsg:= 'FF02 =  Error reaction forced: Non-generative brake order';
	16#FF03: F_AX8xErrMsg:= 'FF03 =  Error reaction forced: Brake chopper off';
	16#FF07: F_AX8xErrMsg:= 'FF07 =  Error reaction forced: Torque Off';
	16#FF08: F_AX8xErrMsg:= 'FF08 =  Error reaction forced: Shorted Coils Brake';
	16#FF09: F_AX8xErrMsg:= 'FF09 =  Error reaction forced: Open Loop Ramp';
	16#FF0A: F_AX8xErrMsg:= 'FF0A =  Error reaction forced: Closed Loop Ramp';
	16#FF0B: F_AX8xErrMsg:= 'FF0B =  Error reaction forced: NC handling';
	16#FF0C: F_AX8xErrMsg:= 'FF0C =  Error reaction TorqueOff with emergency brake';
	16#FFFC: F_AX8xErrMsg:= 'FFFC =  %s';
	16#FFFD: F_AX8xErrMsg:= 'FFFD =  Debug firmware.  Replace "As soon as possible"!';
	16#FFFE: F_AX8xErrMsg:= 'FFFE =  %s';
	16#FFFF: F_AX8xErrMsg:= 'FFFF =  Internal Error.   Additional Errorcode 0x%x';

ELSE
	F_AX8xErrMsg := UINT_TO_STRING(uiDriveError);
	F_AX8xErrMsg := concat(F_AX8xErrMsg, ' Unknown Error code');
END_CASE
F_AX8xErrMsg := F_AX8xErrMsg;

END_FUNCTION

// ---- POUs/FB/FB_2GripperScrewers_New.TcPOU
(*
Nazwa:			FB_2GripperScrewers
Opis:			Zakręcarki szczekowe
Wersja:			v2.62
Data:			2024-10-25
Autor:			DP
Urzadzenia:		Serwo podnośnika, Serwo zakręcania
Ostatnie zmiany:
	- 2024-10-25 [DP] Zmiany torque
	- 2024-08-29 [DP] Wbijak
	- 2024-03-18 [DP] Zmiana symulacji
	- 2024-03-06 [DP] Aktualizacja instrukcji
	- 2024-02-27 [DP] Height Vel z 0 na zadaną w ressetingu, opis problemów
	- 2023-11-24 [DP] Pop. uwag dodatkowych opcji, tryb momentowy - opis
	- 2023-11-10 [DP] Akt. instrukcji, szukanie z UJL
	- 2023-03-25 [DP] przyśpieszenie screwera na stałe, zmiana instrukcji konfiguracji, skrocona czasowka griper
	- 2023-03-21 [DP] dodana ScrewerSet2
	- 2023-02-22 [DP] poprawa w GearRatio
	- 2023-02-21 [DP] Acc, Dec, Jerk i Prędkości Liftera zmniejszone 2x przez inny montaż,
				EStop w StateError, zmiana przekadni obrotu, CycleDone jak SetTorque=0,
	- 2023-02-14 [DP] Zmiana instrukcji konfiguracji
	- 2023-02-14 [DP] Wersja z LU208 z aktualizacjami z XTSa (gearing przy zakręcaniu i szukanie gwintu)
	
Konfiguracja:

Oś Obrótu (AM8031-0C20-0000): 

	Drive:
	- LU207,UBL50 - Nowa zębatka ma 32 na 48 zęby 240:360
	- ustawić driva na 'Rotatory' 360 st. i gear ratio 240:360, 240 st. na obr.
	- Invert Nc-Enc i Nc-Drive włączone
	- włączyć w drivie Scaling->Modulo data storage source - Feeback 1
	- ustawić drive Scaling->position offset setting 0 stopni na odpowiedniej pozycji na enkoderze
	- wgrać z drive Save NC parameters
	- w drivie jeszcze raz ustawić parametr Following error window 359?	
	- ustawic regulator Position mode na Kv na 10, Kp na 0.2, Tn na 0.002 
	- ustawić Acceleration Feed forward  K = 1 i wpisać inercje w Vel contr.->Vel. calc->0.001 kg m^2 oraz Mode->Basic_for_know_interia
	- ustawić w parametrach Configured channel peak current na 5A
	- ustawić w parametrach 0x6072 Bipolar torque/force limit value na 500%
	- ustawić w parametrach 0x60E0 Positive torque/force limit value na 500%
	- ustawić w parametrach 0x60E1 Negative torque/force limit value na 500%
	- dodać parametry Bipolar torque/Force limit w Process data/Outputs i polinkować ze zmienną
	- dodać parametr Positon control proportional gain Process data/Outputs i polinkować ze zmienną
	NC:
	- Ustawić Maximum Velocity na 13397.8, Reference Velocity na 14737.5, Max Acc i Dec na 300000.0
	- Default Acc i Dec na 20096.7, jerk na 60290.0
	- wyłączyć Limity Switche
	- wyłączyć wszystkie opcje Monitoringu

	Opcja trybu momentowego osi zakręcania (tylko od wersji driva 104)
	Drvie:
	- Na jednym drivie nie może być razem obrót 1 i obrót 2
	- W drivie (kanał) osi obrotu Advanced->Slots settings zaznaczyć 'I know what I do'
	i ustawiąc VelocityControlSlot na VelocityControl2, w tym momencie w IO powinny pojawić się 
	nowe wejścia,wyjścia VelocityControl2
	- W drivie Advanced->Process data rozwinąć 'Ch A Modes of operation' i ustawić '..mode_CST (10)'
	w Virual operation mode 0 
	- W parametr list powinien być parametr 0x60CA Ch a Torque limitation option code -> ustwić na
	TorqueMightBeReducedToZero, jeżeli nie ma to znaczy że trzeba zaktualizować driva lub dodać parametry ręcznie
	NC:
	- W NC w Drive->Zakładka Time Comensation-> Parametr Time Compensation Mode Drive -> 'ON(with velocity)'
	- W NC w Enc->Zakładka Time Comensation-> Parametr Time Compensation Mode Drive -> 'ON(with velocity)'
	
Oś podnoszenia (AM8032-0E21-0000):
	Drive:
	- ustawić driva na 'Linerary' 10mm i gear ratio 1:1, 10mm na obr.
	- Invert Nc-Enc i Nc-Drive włączone
	- ustawic regulator Position mode na Kv na 1, Kp na 0.2, Tn na 0.002 
	- ustawić Feed forward acceleration K = 1 i wpisać inercje w Vel contr.->Cel. calc->0 kg m^2
	NC:
	- Ustawić Maximum Velocity na 1094
	- Default Acc i Dec na 100000, jerk na 500000
	- ustawić Limit Swtiche
	- ustawić ManualVelocity (Slow) na 30 ze względu na Jog i bazowanie

Info: 
	- możliwość pracy 1 lub 2
	- możliwość pracy bez kręcenia jeżeli ustawi się prędkość 0
	- możliwosć dodatkowego chwytania przed zakręcaniem
	- step mode dla wizualizacji
	- rozróżnienie warningów

Tryb momementowy:
lrPackageTurnoversToFullScrewed - Ilośc obrotów do zakręcenia
iScrewer1SetTorque - Zadany moment w % (Przeliczany z Nm z wizualizacji)
lrScrewerSpeed - Prędkość zakręcania w st/s (Przeliczany z rpm z wizualziacji)
1. Start											Rozpędzanie,	Torque 5000 (Max) [%], 				TorqueRamp 4000 [%/s], VelocityLimitLow -5000 (Max) [st./s]
2. ActPos>lrPackageTurnoversToFullScrewed*360.0/7	Hamowanie,		Torque -9 [%],						TorqueRamp 1500 [%/s], VelocityLimitLow -4000 (Max) [st./s]
3. ActPos>lrPackageTurnoversToFullScrewed*360.0/6	Dokręcanie,		Torque iScrewer1SetTorque [%],		TorqueRamp 4000 [%/s], VelocityLimitLow lrScrewerSpeed (Max) [st./s]



Jak naprawić:
A. Zakręcarka nie wykonuje ruchu w trybie momentowym, jedna działa , druga nie - sprawdzić czy bloczek MC_Torque wykonuje ruchu,
jeżeli nie to wyłączyć VelocityControl2, włączyć bez '2' i ponownie włączyć '2', potem aktywacja
B. 
*)

FUNCTION_BLOCK FB_2GripperScrewers_New
VAR_INPUT
	bEnable1							:BOOL;		//Zezwolenie na pracę 1
	bEnable2							:BOOL;		//Zezwolenie na pracę 2
	bEstop								:BOOL;		//Stop awaryjny nieaktywny
	bRun1								:BOOL;		//Rozkaz zakręcania zakręcarki 1
	bRun2								:BOOL;		//Rozkaz zakręcania zakręcarki 2
	bSimulation							:BOOL;		//Włączona symulacja, skracanie czasu przerywania jak nie ma butelki
	bHoming								:BOOL;		//Zezwolenie na wykonanie bazowania i pozycjonowania zakręcarki
	bHeightSet							:BOOL;		//Ustaw wysokość
	bIgnoreError						:BOOL;		//Ignorowania błędów cyklu pracy
	bScrewer1SetPositionOffset			:BOOL;		//Ustaw offset obrotu zakręcarki 1
	bScrewer2SetPositionOffset			:BOOL;		//Ustaw offset obrotu zakręcarki 2
	iScrewer1AddTorque					:UINT;
	iScrewer2AddTorque					:UINT;
	bReset								:BOOL;		//Reset błędu, jeśli w stanie "eError
	iTool								:INT;		// Wybór narzędzia (1-5), opisy w tablicy AsGripperScrewerTool	
	bOptionOpenedGripperWhenFindingScrew:BOOL;		//OPCJA. Otwarty chwytak przy szukaniu gwintu
	bOptionScrewingBackwardsInPushingPosition:BOOL;	//OPCJA. Obrót do tyłu w pozycji dociskania
	bOptionCapPushingWithoutScrewing	:BOOL;		//OPCJA. Tylko wbijanie bez zakręcania
	bOptionCapPositioning				:BOOL;		//OPCJA. Dodatkowe zamknięcie chwytakiem przed zakręceniem (do testów)
	bOptionFindScrewInScrewingPosition	:BOOL;		//OPCJA. Szukaj początku gwintu nakrętki i opakowania. Zakręcarka napjpierw obraca się w lewo, a po znalezienu gwintu przystepuje do zakręcania w pozycji zakręcania
	bOptionFindScrewInPushingPosition	:BOOL;		//OPCJA. Szukaj początku gwintu nakrętki i opakowania. Zakręcarka napjpierw obraca się w lewo, a po znalezienu gwintu przystepuje do zakręcania w pozycsji docisku
	bOptionFindScrewWithHeightSensor	:BOOL;		//OPCJA. Szukanie gwintu z czujnikiem wysokości
	bOptionFindScrewRotateFromPushingToScrewingSensor	:BOOL;		//OPCJA. Obrót od pozycji docisku do zakręcania
	bOptionMomentaryMode				:BOOL;		//OPCJA. Tryb momentowy zakręcania
	lrPackageTurnoversToFullScrewed		:LREAL;		//Obroty do pełnego zakręcenia
	lrPackageThreadPitch				:LREAL;		//Skok gwintu
	lrPackageThreadTimes				:LREAL;		//Krotność gwintu
	lrHeightReadyPosition				:LREAL;		//Wysokość zadana w stanie gotowości od płyty[mm]
	lrHeightPushingPosition				:LREAL;		//Wysokość zadana przy wciskaniu nakrętki od płyty[mm]
	lrHeightEndScrewingPosition			:LREAL;		//Wysokość zadana przy zakręcaniu nakrętki od płyty [mm]
	lrHeightScrewingDistanceSpeed		:REAL;		//Prędkość obniżania podczas zakręcania
	lrHeightActualPosition				:LREAL;		//Aktualna pozycja podnośnika
	diSensorHeightCV					:DINT;		//Czujnik wysokości IO-Link
	rSensorHeightCV						:REAL;		//Czujnik wysokości IO-Link w mm
	lrHeightActualTorque				:LREAL;		//Aktualny moment [%]
	rActualMotor1Temperature			:REAL;		//Aktualna temperatura silnika 1
	rActualMotor2Temperature			:REAL;		//Aktualna temperatura silnika 2
	iHeightSetTorque					:INT;		//Zadany moment dociskania [%]
	iScrewer1SetTorque					:INT;		//Zadany moment dokręcania [%]
	iScrewer2SetTorque					:INT;		//Zadany moment dokręcania [%]
	iScrewTightTime						:INT;		//Czas przytrzymania po uzyskaniu momentu [ms] 
	lrScrewer1ActualTorque				:LREAL;		//Aktualny moment [%]
	lrScrewer2ActualTorque				:LREAL;		//Aktualny moment [%]
	lrHeightAcceleration				:LREAL;		//Przyspieszenie podnosnika zakręcarki
	lrHeightDeceleration				:LREAL;		//Opóźnienie podnośnika zakręcarki
	lrHeightSpeed						:LREAL;		//Prędkość podnośnika zakręcarki
	lrScrewer1ActualPosition			:LREAL;	
	lrScrewer2ActualPosition			:LREAL;	
	lrScrewerAcceleration				:LREAL;		//Przyspieszenie zakręcania
	lrScrewerDeceleration				:LREAL;		//Opóźnienie zakręcania
	lrScrewerSpeed						:LREAL;		//Prędkość zakręcania
	lrScrewer1PosDiff					:LREAL;		//ScrewingAxisRef.NcToPlc.PosDiff
	lrScrewer2PosDiff					:LREAL;		//ScrewingAxisRef.NcToPlc.PosDiff
	lrFindigScrewDegree					:LREAL;		//Kąt wycofania zakręcarki przy szukaniu gwintu
	bManualMovement						:BOOL;		//Zezwolenie na ruchy ręcznę
	lrManualOverride					:LREAL;		//Procentowa redukcja prędkości wszystkich serw (Tylko w trybie manualnym)
                                	
	lrMaxHeightPosition:LREAL;				//Wysokość maksymalna zakręcarki 
	lrMinHeightPosition:LREAL;				//Wysokość minimalna zakręcarki 
	lrMaxScrewerSpeed	:LREAL;				//Maksymalna prędkość zakręcania

	//StepMode
	bStepMode				: BOOL;		//Włączony tryb skokowy sterowania podnośnikami (tylko w serwisie)
	lrSetPosStepMode		: LREAL; 	//Ruch podnośnika o zadaną wartość w trybie krokowym (tylko w serwisie)
	
	_ALARMINFO_ :BOOL;
	iStationIndex:UDINT;					//Numer stacji 
	sStationName:STRING;					//Nazwa stacji
END_VAR

VAR_OUTPUT
	eState							: E_Station;				//Stan ogólny bloku
	eRunningState					: E_GripperScrewer; 		//Stan zakręcarki
	bError							: BOOL;						//Błąd stacji
	udiErrorID						: UDINT;					//Nr błędu zakręcarki
	sErrorDescription				: STRING(200);				//Opis błędu
	sErrorDescription2				: STRING(200);				//Opis błędu
	sErrorStationName				: STRING;					//Nazwa stacj
	udiStationID					: UDINT;				// Nr stacji
	
	udiHeightServoErrorNr			: UDINT;					//Nr błędu serwo podnośnika
	udiScrewing1ServoErrorNr		: UDINT;					//Nr błędu serwo zakręcarki 1
	udiScrewing2ServoErrorNr		: UDINT;					//Nr błędu serwo zakręcarki 2
	udiScrewing1EncoderErrorNr		: UDINT;					//Nr błędu encodera zakręcarki 1
	bGripper1Actuator				: BOOL;						//Siłownik chwytaka
	bGripper2Actuator				: BOOL;						//Siłownik chwytaka
	uiScrewing1TorqueControl		: UINT;						//Kontola momentu zakręcania	
	uiScrewing2TorqueControl		: UINT;						//Kontola momentu zakręcania	
	rScrewing1ProportionalGain		: UINT;						//Kontola Kp
	rScrewing2ProportionalGain		: UINT;						//Kontola Kp	
	lrScrewer1TorqueCV				: LREAL;					//Wartość osiągniętego momentu dokręcenia [nM]
	lrScrewer2TorqueCV				: LREAL;					//Wartość osiągniętego momentu dokręcenia [nM]
	uiHeightTorqueControl			: UINT						:= 6000;
	sWarningDescription				: STRING;
	bWarning1						: BOOL;
	bWarning1A						: BOOL;	
	bWarning1B						: BOOL;	
	bWarning1C						: BOOL;	
	bWarning1D						: BOOL;	
	bWarning1E						: BOOL;	{warning'dorobic ostrzezenie szukania gwintu}
	bWarning2						: BOOL;
	bWarning2A						: BOOL;	
	bWarning2B						: BOOL;	
	bWarning2C						: BOOL;	
	bWarning2D						: BOOL;	
	bWarning2E						: BOOL;	
	udiWarningID					: UDINT;
	tCycleTime						: TIME;	
	bHomingDone						: BOOL;						//Wymagane ponowne bazowanie (blad podczas bazowania lub stop awaryjny)
	bCycleDone1						: BOOL;
	bCycleNotDone1					: BOOL;		
	bCycleDone2						: BOOL;
	bCycleNotDone2					: BOOL;		
	bAdjustingTorqueDone			: BOOL;
	iAdjustingTorque				: INT;
	lrAdjustingMaxTorque			: LREAL;
	AsToolDescription				: ARRAY [0..10] OF STRING;	// Opis narzędzi, 1 - Opis narzędzia nr 1, 2 - Opis narzędzia nr 2
	sTool							: STRING;
END_VAR

VAR_IN_OUT
	bManualHeightUp					:BOOL;			//Ruch ręczny podnośnikiem stacji w górę
	bManualHeightDown				:BOOL;			//Ruch ręczny podnośnikiem stacji w dół
	bManualScrew1Clockwise			:BOOL;			//Ruch ręczny zakręcarką w kierunku wskazówek zegara;
	bManualScrew1CClockwise			:BOOL;			//Ruch ręczny zakręcarką w kierunku przeciwnym do wskazówek zegara;
	bManualScrew2Clockwise			:BOOL;			//Ruch ręczny zakręcarką w kierunku wskazówek zegara;
	bManualScrew2CClockwise			:BOOL;			//Ruch ręczny zakręcarką w kierunku przeciwnym do wskazówek zegara;
	bManualGripper1					:BOOL;			//Ruch zamknięcie chwytaka nakrętek
	bManualGripper2					:BOOL;			//Ruch zamknięcie chwytaka nakrętek
	HeightAxisRef					:AXIS_REF;		//Struktura sterowania NC dla serwa podnoszenia zakręcarki
	Screwing1AxisRef				:AXIS_REF;		//Struktura sterowania NC dla serwa zakręcania
	Screwing2AxisRef				:AXIS_REF;		//Struktura sterowania NC dla serwa zakręcania	
	Screwing1EncoderAxisRef			:AXIS_REF;		//Struktura sterowania NC dla serwa zakręcania
	bFindScrewAdjustSensorHeight	:BOOL;			//Włacz szukanie MIN i MAX jeżeli jest opcja z czujnikie wysokości
	bAdjustingTorque				:BOOL;			//Dobieranie momentu
	lrAdjustingSetTorque			:LREAL;	
END_VAR

VAR
	bScrew1Found					: BOOL; 						// Zakręcarka znalazła początek gwintu
	bScrew2Found					: BOOL; 						// Zakręcarka znalazła początek gwintu	
	tonTightScrewing1Timer			: TON; 							// Timer potwierdzenia dokręcenia nakrętki
	tonTightScrewing2Timer			: TON; 							// Timer potwierdzenia dokręcenia nakrętki
	tonTightScrewing1TimerAndOpenedGripper	: TON; 					// Timer potwierdzenia dokręcenia nakrętki
	tonTightScrewing2TimerAndOpenedGripper	: TON; 					// Timer potwierdzenia dokręcenia nakrętki	
	tonMomentaryScrewing1Timer		: TON; 							// Timer potwierdzenia dokręcenia nakrętki
	tonMomentaryScrewing2Timer		: TON; 							// Timer potwierdzenia dokręcenia nakrętki

	bScrewed1					: BOOL; 						// Nakrętka zakręcona
	bScrewed2					: BOOL; 						// Nakrętka zakręcona
	tonTooLongScrewing1			: TON;							// Błąd zbyt długiego zakręcania
	tonTooLongScrewing2			: TON; 							// Błąd zbyt długiego zakręcania	
	tTooLongScrewing1			: TIME;							// Czas  zbyt długiego zakręcania
	tTooLongScrewing2			: TIME; 						// Czas  zbyt długiego zakręcania		
	tonGripper1ReliseDelay		: TON;							// Time Opóźniajacy ruch w górę po zakręceniu, pozwalajac na otwarcie chwytaka
	tonGripper2ReliseDelay		: TON;							// Time Opóźniajacy ruch w górę po zakręceniu, pozwalajac na otwarcie chwytaka
	tonGripper1ReliseDelay2		: TON;							// Time Opóźniajacy ruch w górę po zakręceniu, pozwalajac na otwarcie chwytaka
	tonGripper2ReliseDelay2		: TON;							// Time Opóźniajacy ruch w górę po zakręceniu, pozwalajac na otwarcie chwytaka

	mcScrewer1ManualMove		: MC_JOG; 						// Blok obrotu ręcznego zakręcarką
	mcScrewer2ManualMove		: MC_JOG; 						// Blok obrotu ręcznego zakręcarką
	mcScrewer1Stop				: MC_Stop;						// Trwałe zatrzymywanie Serwo
	mcScrewer2Stop				: MC_Stop;						// Trwałe zatrzymywanie Serwo
	mcScrewer1MoveVelocity		: MC_MoveVelocity;				// Ruch prędkościowy
	mcScrewer2MoveVelocity		: MC_MoveVelocity;				// Ruch prędkościowy
	mcScrewer1MoveVelocity2		: MC_MoveVelocity;				// Ruch prędkościowy
	mcScrewer2MoveVelocity2		: MC_MoveVelocity;				// Ruch prędkościowy
	mcScrewer1MoveVelocity3		: MC_MoveVelocity;				// Ruch prędkościowy
	mcScrewer2MoveVelocity3		: MC_MoveVelocity;				// Ruch prędkościowy	
	mcScrewer1MoveRelative		: MC_MoveRelative; 				// Ruch relatywny zakręcarki
	mcScrewer2MoveRelative		: MC_MoveRelative; 				// Ruch relatywny zakręcarki
	mcScrewer1MoveAbsolute		: MC_MoveAbsolute; 				// Ruch absolutny zakręcarki
	mcScrewer2MoveAbsolute		: MC_MoveAbsolute; 				// Ruch absolutny zakręcarki
	fbScrewer1SetPositionOffset	: FB_CoEAX8000SetPositionOffset;// Ustawianie pozycji obrotu 
	fbScrewer2SetPositionOffset	: FB_CoEAX8000SetPositionOffset;// Ustawianie pozycji obrotu 
	mcScrewer1TorqueControl		: MC_TorqueControl;
	mcScrewer2TorqueControl		: MC_TorqueControl;
	
	mcScrewer1MoveContinuousRel	: MC_MoveContinuousRelative;
	mcScrewer2MoveContinuousRel	: MC_MoveContinuousRelative;
	
